gfCNCPoint4[20422] = {X 336.3907, Y 58.0000, Z -6.3333, A 0.000, B 0.000, C 0.000 }
gfCNCPoint4[20423] = {X 336.3907, Y 58.9517, Z -6.3333, A 0.000, B 0.000, C 0.000 }
gfCNCPoint4[20424] = {X 336.3894, Y 59.0936, Z -6.3333, A 0.000, B 0.000, C 0.000 }
gfCNCPoint4[20425] = {X 336.3864, Y 59.2354, Z -6.3333, A 0.000, B 0.000, C 0.000 }
gfCNCPoint4[20426] = {X 336.2429, Y 60.7995, Z -6.3333, A 0.000, B 0.000, C 0.000 }
gfCNCPoint4[20427] = {X 335.8982, Y 62.3319, Z -6.3333, A 0.000, B 0.000, C 0.000 }
gfCNCPoint4[20428] = {X 335.3582, Y 63.8069, Z -6.3333, A 0.000, B 0.000, C 0.000 }
gfCNCPoint4[20429] = {X 334.6320, Y 65.1996, Z -6.3333, A 0.000, B 0.000, C 0.000 }
gfCNCPoint4[20430] = {X 333.7317, Y 66.4867, Z -6.3333, A 0.000, B 0.000, C 0.000 }
gfCNCPoint4[20431] = {X 332.6725, Y 67.6465, Z -6.3333, A 0.000, B 0.000, C 0.000 }
gfCNCPoint4[20432] = {X 332.6738, Y 81.6369, Z -6.3333, A 0.000, B 0.000, C 0.000 }
gfCNCPoint4[20433] = {X 334.6671, Y 81.9567, Z -6.3333, A 0.000, B 0.000, C 0.000 }
gfCNCPoint4[20434] = {X 336.6742, Y 82.1743, Z -6.3333, A 0.000, B 0.000, C 0.000 }
gfCNCPoint4[20435] = {X 340.8156, Y 82.4531, Z -6.3333, A 0.000, B 0.000, C 0.000 }
gfCNCPoint4[20436] = {X 344.9638, Y 82.5981, Z -6.3333, A 0.000, B 0.000, C 0.000 }
gfCNCPoint4[20437] = {X 349.1145, Y 82.6093, Z -6.3333, A 0.000, B 0.000, C 0.000 }
gfCNCPoint4[20438] = {X 353.0020, Y 82.5472, Z -6.3333, A 0.000, B 0.000, C 0.000 }
gfCNCPoint4[20439] = {X 356.8847, Y 82.3434, Z -6.3333, A 0.000, B 0.000, C 0.000 }
gfCNCPoint4[20440] = {X 360.7573, Y 81.9982, Z -6.3333, A 0.000, B 0.000, C 0.000 }
gfCNCPoint4[20441] = {X 361.9619, Y 81.8410, Z -6.3333, A 0.000, B 0.000, C 0.000 }
gfCNCPoint4[20442] = {X 363.1593, Y 81.6353, Z -6.3333, A 0.000, B 0.000, C 0.000 }
gfCNCPoint4[20443] = {X 363.1584, Y 67.6531, Z -6.3333, A 0.000, B 0.000, C 0.000 }
gfCNCPoint4[20444] = {X 362.0724, Y 66.4629, Z -6.3333, A 0.000, B 0.000, C 0.000 }
gfCNCPoint4[20445] = {X 361.1545, Y 65.1387, Z -6.3333, A 0.000, B 0.000, C 0.000 }
gfCNCPoint4[20446] = {X 360.4210, Y 63.7042, Z -6.3333, A 0.000, B 0.000, C 0.000 }
gfCNCPoint4[20447] = {X 359.8849, Y 62.1848, Z -6.3333, A 0.000, B 0.000, C 0.000 }
gfCNCPoint4[20448] = {X 359.5557, Y 60.6075, Z -6.3333, A 0.000, B 0.000, C 0.000 }
gfCNCPoint4[20449] = {X 359.4395, Y 59.0005, Z -6.3333, A 0.000, B 0.000, C 0.000 }
gfCNCPoint4[20450] = {X 359.4393, Y 58.0000, Z -6.3333, A 0.000, B 0.000, C 0.000 }
gfCNCPoint4[20451] = {X 359.5340, Y 56.4902, Z -6.3333, A 0.000, B 0.000, C 0.000 }
gfCNCPoint4[20452] = {X 359.8167, Y 55.0040, Z -6.3333, A 0.000, B 0.000, C 0.000 }
gfCNCPoint4[20453] = {X 359.6068, Y 55.1023, Z -6.3333, A 0.000, B 0.000, C 0.000 }
gfCNCPoint4[20454] = {X 359.3961, Y 55.1989, Z -6.3333, A 0.000, B 0.000, C 0.000 }
gfCNCPoint4[20455] = {X 357.8730, Y 55.8158, Z -6.3333, A 0.000, B 0.000, C 0.000 }
gfCNCPoint4[20456] = {X 356.3192, Y 56.3507, Z -6.3333, A 0.000, B 0.000, C 0.000 }
gfCNCPoint4[20457] = {X 353.9698, Y 56.9888, Z -6.3333, A 0.000, B 0.000, C 0.000 }
gfCNCPoint4[20458] = {X 351.5774, Y 57.4394, Z -6.3333, A 0.000, B 0.000, C 0.000 }
gfCNCPoint4[20459] = {X 349.1568, Y 57.6995, Z -6.3333, A 0.000, B 0.000, C 0.000 }
gfCNCPoint4[20460] = {X 348.9949, Y 55.3050, Z -6.3333, A 0.000, B 0.000, C 0.000 }
gfCNCPoint4[20461] = {X 348.0810, Y 55.3520, Z -6.3333, A 0.000, B 0.000, C 0.000 }
gfCNCPoint4[20462] = {X 347.1660, Y 55.3695, Z -6.3333, A 0.000, B 0.000, C 0.000 }
gfCNCPoint4[20463] = {X 344.5859, Y 55.3176, Z -6.3333, A 0.000, B 0.000, C 0.000 }
gfCNCPoint4[20464] = {X 342.0205, Y 55.0380, Z -6.3333, A 0.000, B 0.000, C 0.000 }
gfCNCPoint4[20465] = {X 339.4899, Y 54.5327, Z -6.3333, A 0.000, B 0.000, C 0.000 }
gfCNCPoint4[20466] = {X 337.0138, Y 53.8057, Z -6.3333, A 0.000, B 0.000, C 0.000 }
gfCNCPoint4[20467] = {X 334.7570, Y 52.9268, Z -6.3333, A 0.000, B 0.000, C 0.000 }
gfCNCPoint4[20468] = {X 332.5808, Y 51.8637, Z -6.3333, A 0.000, B 0.000, C 0.000 }
gfCNCPoint4[20469] = {X 331.5853, Y 51.2779, Z -6.3333, A 0.000, B 0.000, C 0.000 }
gfCNCPoint4[20470] = {X 330.6137, Y 50.6533, Z -6.3333, A 0.000, B 0.000, C 0.000 }
gfCNCPoint4[20471] = {X 331.5795, Y 51.6073, Z -6.3333, A 0.000, B 0.000, C 0.000 }
gfCNCPoint4[20472] = {X 332.4023, Y 52.6870, Z -6.3333, A 0.000, B 0.000, C 0.000 }
gfCNCPoint4[20473] = {X 333.0660, Y 53.8713, Z -6.3333, A 0.000, B 0.000, C 0.000 }
gfCNCPoint4[20474] = {X 333.5575, Y 55.1367, Z -6.3333, A 0.000, B 0.000, C 0.000 }
gfCNCPoint4[20475] = {X 333.8672, Y 56.4585, Z -6.3333, A 0.000, B 0.000, C 0.000 }
gfCNCPoint4[20476] = {X 333.9598, Y 57.2268, Z -6.3333, A 0.000, B 0.000, C 0.000 }
gfCNCPoint4[20477] = {X 333.9907, Y 58.0000, Z -6.3333, A 0.000, B 0.000, C 0.000 }
gfCNCPoint4[20478] = {X 333.9907, Y 58.9439, Z -6.3333, A 0.000, B 0.000, C 0.000 }
gfCNCPoint4[20479] = {X 333.8763, Y 60.3992, Z -6.3333, A 0.000, B 0.000, C 0.000 }
gfCNCPoint4[20480] = {X 333.5452, Y 61.8209, Z -6.3333, A 0.000, B 0.000, C 0.000 }
gfCNCPoint4[20481] = {X 333.0049, Y 63.1770, Z -6.3333, A 0.000, B 0.000, C 0.000 }
gfCNCPoint4[20482] = {X 332.2676, Y 64.4368, Z -6.3333, A 0.000, B 0.000, C 0.000 }
gfCNCPoint4[20483] = {X 331.3498, Y 65.5720, Z -6.3333, A 0.000, B 0.000, C 0.000 }
gfCNCPoint4[20484] = {X 330.2724, Y 66.5569, Z -6.3333, A 0.000, B 0.000, C 0.000 }
gfCNCPoint4[20485] = {X 330.2739, Y 83.2031, Z -6.3333, A 0.000, B 0.000, C 0.000 }
gfCNCPoint4[20486] = {X 330.2776, Y 83.5824, Z -6.3333, A 0.000, B 0.000, C 0.000 }
gfCNCPoint4[20487] = {X 333.3587, Y 84.1905, Z -6.3333, A 0.000, B 0.000, C 0.000 }
gfCNCPoint4[20488] = {X 336.4766, Y 84.5661, Z -6.3333, A 0.000, B 0.000, C 0.000 }
gfCNCPoint4[20489] = {X 340.6882, Y 84.8497, Z -6.3333, A 0.000, B 0.000, C 0.000 }
gfCNCPoint4[20490] = {X 344.9068, Y 84.9975, Z -6.3333, A 0.000, B 0.000, C 0.000 }
gfCNCPoint4[20491] = {X 349.1279, Y 85.0093, Z -6.3333, A 0.000, B 0.000, C 0.000 }
gfCNCPoint4[20492] = {X 353.0977, Y 84.9454, Z -6.3333, A 0.000, B 0.000, C 0.000 }
gfCNCPoint4[20493] = {X 357.0624, Y 84.7369, Z -6.3333, A 0.000, B 0.000, C 0.000 }
gfCNCPoint4[20494] = {X 361.0169, Y 84.3841, Z -6.3333, A 0.000, B 0.000, C 0.000 }
gfCNCPoint4[20495] = {X 363.3029, Y 84.0502, Z -6.3333, A 0.000, B 0.000, C 0.000 }
gfCNCPoint4[20496] = {X 365.5594, Y 83.5549, Z -6.3333, A 0.000, B 0.000, C 0.000 }
gfCNCPoint4[20497] = {X 365.5583, Y 66.5610, Z -6.3333, A 0.000, B 0.000, C 0.000 }
gfCNCPoint4[20498] = {X 364.4841, Y 65.5830, Z -6.3333, A 0.000, B 0.000, C 0.000 }
gfCNCPoint4[20499] = {X 363.5683, Y 64.4553, Z -6.3333, A 0.000, B 0.000, C 0.000 }
gfCNCPoint4[20500] = {X 362.8315, Y 63.2032, Z -6.3333, A 0.000, B 0.000, C 0.000 }
gfCNCPoint4[20501] = {X 362.2905, Y 61.8550, Z -6.3333, A 0.000, B 0.000, C 0.000 }
gfCNCPoint4[20502] = {X 361.9573, Y 60.4410, Z -6.3333, A 0.000, B 0.000, C 0.000 }
gfCNCPoint4[20503] = {X 361.8395, Y 58.9930, Z -6.3333, A 0.000, B 0.000, C 0.000 }
gfCNCPoint4[20504] = {X 361.8393, Y 58.0000, Z -6.3333, A 0.000, B 0.000, C 0.000 }
gfCNCPoint4[20505] = {X 361.9152, Y 56.7901, Z -6.3333, A 0.000, B 0.000, C 0.000 }
gfCNCPoint4[20506] = {X 362.1417, Y 55.5992, Z -6.3333, A 0.000, B 0.000, C 0.000 }
gfCNCPoint4[20507] = {X 362.5727, Y 54.3039, Z -6.3333, A 0.000, B 0.000, C 0.000 }
gfCNCPoint4[20508] = {X 363.1817, Y 53.0820, Z -6.3333, A 0.000, B 0.000, C 0.000 }
gfCNCPoint4[20509] = {X 363.9565, Y 51.9580, Z -6.3333, A 0.000, B 0.000, C 0.000 }
gfCNCPoint4[20510] = {X 364.8817, Y 50.9541, Z -6.3333, A 0.000, B 0.000, C 0.000 }
gfCNCPoint4[20511] = {X 365.9389, Y 50.0904, Z -6.3333, A 0.000, B 0.000, C 0.000 }
gfCNCPoint4[20512] = {X 367.1071, Y 49.3840, Z -6.3333, A 0.000, B 0.000, C 0.000 }
gfCNCPoint4[20513] = {X 368.3631, Y 48.8490, Z -6.3333, A 0.000, B 0.000, C 0.000 }
gfCNCPoint4[20514] = {X 369.6819, Y 48.4960, Z -6.3333, A 0.000, B 0.000, C 0.000 }
gfCNCPoint4[20515] = {X 371.0372, Y 48.3320, Z -6.3333, A 0.000, B 0.000, C 0.000 }
gfCNCPoint4[20516] = {X 371.2782, Y 48.3230, Z -6.3333, A 0.000, B 0.000, C 0.000 }
gfCNCPoint4[20517] = {X 371.5193, Y 48.3200, Z -6.3333, A 0.000, B 0.000, C 0.000 }
gfCNCPoint4[20518] = {X 388.0597, Y 48.3200, Z -6.3333, A 0.000, B 0.000, C 0.000 }
gfCNCPoint4[20519] = {X 389.4419, Y 48.4192, Z -6.3333, A 0.000, B 0.000, C 0.000 }
gfCNCPoint4[20520] = {X 390.7958, Y 48.7147, Z -6.3333, A 0.000, B 0.000, C 0.000 }
gfCNCPoint4[20521] = {X 392.0936, Y 49.2006, Z -6.3333, A 0.000, B 0.000, C 0.000 }
gfCNCPoint4[20522] = {X 393.3087, Y 49.8667, Z -6.3333, A 0.000, B 0.000, C 0.000 }
gfCNCPoint4[20523] = {X 394.5333, Y 49.1962, Z -6.3333, A 0.000, B 0.000, C 0.000 }
gfCNCPoint4[20524] = {X 395.8416, Y 48.7089, Z -6.3333, A 0.000, B 0.000, C 0.000 }
gfCNCPoint4[20525] = {X 397.1858, Y 48.4177, Z -6.3333, A 0.000, B 0.000, C 0.000 }
gfCNCPoint4[20526] = {X 398.5577, Y 48.3200, Z -6.3333, A 0.000, B 0.000, C 0.000 }
gfCNCPoint4[20527] = {X 398.7346, Y 48.3200, Z -6.3333, A 0.000, B 0.000, C 0.000 }
gfCNCPoint4[20528] = {X 398.1859, Y 47.6069, Z -6.3333, A 0.000, B 0.000, C 0.000 }
gfCNCPoint4[20529] = {X 397.7774, Y 46.8051, Z -6.3333, A 0.000, B 0.000, C 0.000 }
gfCNCPoint4[20530] = {X 397.5230, Y 45.9420, Z -6.3333, A 0.000, B 0.000, C 0.000 }
gfCNCPoint4[20531] = {X 397.4561, Y 45.4921, Z -6.3333, A 0.000, B 0.000, C 0.000 }
gfCNCPoint4[20532] = {X 397.4314, Y 45.0378, Z -6.3333, A 0.000, B 0.000, C 0.000 }
gfCNCPoint4[20533] = {X 397.4316, Y 44.1456, Z -6.3333, A 0.000, B 0.000, C 0.000 }
gfCNCPoint4[20534] = {X 397.5413, Y 43.1780, Z -6.3333, A 0.000, B 0.000, C 0.000 }
gfCNCPoint4[20535] = {X 397.8410, Y 42.2514, Z -6.3333, A 0.000, B 0.000, C 0.000 }
gfCNCPoint4[20536] = {X 398.3186, Y 41.4029, Z -6.3333, A 0.000, B 0.000, C 0.000 }
gfCNCPoint4[20537] = {X 398.9552, Y 40.6660, Z -6.3333, A 0.000, B 0.000, C 0.000 }
gfCNCPoint4[20538] = {X 398.9552, Y 31.8248, Z -6.3333, A 0.000, B 0.000, C 0.000 }
gfCNCPoint4[20539] = {X 396.7504, Y 27.9907, Z -6.3333, A 0.000, B 0.000, C 0.000 }
gfCNCPoint4[20540] = {X 386.3478, Y 33.9728, Z -6.3333, A 0.000, B 0.000, C 0.000 }
gfCNCPoint4[20541] = {X 386.2674, Y 34.3975, Z -6.3333, A 0.000, B 0.000, C 0.000 }
gfCNCPoint4[20542] = {X 386.1833, Y 34.8215, Z -6.3333, A 0.000, B 0.000, C 0.000 }
gfCNCPoint4[20543] = {X 386.0240, Y 35.5723, Z -6.3333, A 0.000, B 0.000, C 0.000 }
gfCNCPoint4[20544] = {X 385.8510, Y 36.3200, Z -6.3333, A 0.000, B 0.000, C 0.000 }
gfCNCPoint4[20545] = {X 386.9552, Y 36.3200, Z -6.3333, A 0.000, B 0.000, C 0.000 }
gfCNCPoint4[20546] = {X 386.9552, Y 35.0290, Z -6.3333, A 0.000, B 0.000, C 0.000 }
gfCNCPoint4[20547] = {X 386.3478, Y 33.9728, Z -6.3333, A 0.000, B 0.000, C 0.000 }
gfCNCPoint4[20548] = {X 388.4283, Y 32.7764, Z -6.3333, A 0.000, B 0.000, C 0.000 }
gfCNCPoint4[20549] = {X 384.7454, Y 26.3718, Z -6.3333, A 0.000, B 0.000, C 0.000 }
gfCNCPoint4[20550] = {X 384.6159, Y 28.7722, Z -6.3333, A 0.000, B 0.000, C 0.000 }
gfCNCPoint4[20551] = {X 384.3631, Y 31.1627, Z -6.3333, A 0.000, B 0.000, C 0.000 }
gfCNCPoint4[20552] = {X 383.9877, Y 33.5370, Z -6.3333, A 0.000, B 0.000, C 0.000 }
gfCNCPoint4[20553] = {X 383.9112, Y 33.9411, Z -6.3333, A 0.000, B 0.000, C 0.000 }
gfCNCPoint4[20554] = {X 383.8312, Y 34.3445, Z -6.3333, A 0.000, B 0.000, C 0.000 }
gfCNCPoint4[20555] = {X 383.6810, Y 35.0524, Z -6.3333, A 0.000, B 0.000, C 0.000 }
gfCNCPoint4[20556] = {X 383.5178, Y 35.7575, Z -6.3333, A 0.000, B 0.000, C 0.000 }
gfCNCPoint4[20557] = {X 383.1278, Y 37.2469, Z -6.3333, A 0.000, B 0.000, C 0.000 }
gfCNCPoint4[20558] = {X 382.6801, Y 38.7200, Z -6.3333, A 0.000, B 0.000, C 0.000 }
gfCNCPoint4[20559] = {X 388.0597, Y 38.7200, Z -6.3333, A 0.000, B 0.000, C 0.000 }
gfCNCPoint4[20560] = {X 388.4821, Y 38.7246, Z -6.3333, A 0.000, B 0.000, C 0.000 }
gfCNCPoint4[20561] = {X 388.9042, Y 38.7385, Z -6.3333, A 0.000, B 0.000, C 0.000 }
gfCNCPoint4[20562] = {X 389.1203, Y 38.2363, Z -6.3333, A 0.000, B 0.000, C 0.000 }
gfCNCPoint4[20563] = {X 389.3552, Y 37.7426, Z -6.3333, A 0.000, B 0.000, C 0.000 }
gfCNCPoint4[20564] = {X 389.3552, Y 34.3882, Z -6.3333, A 0.000, B 0.000, C 0.000 }
gfCNCPoint4[20565] = {X 388.4283, Y 32.7764, Z -6.3333, A 0.000, B 0.000, C 0.000 }
gfCNCPoint4[20566] = {X 390.5088, Y 31.5799, Z -6.3333, A 0.000, B 0.000, C 0.000 }
gfCNCPoint4[20567] = {X 386.7932, Y 25.1185, Z -6.3333, A 0.000, B 0.000, C 0.000 }
gfCNCPoint4[20568] = {X 386.1529, Y 24.0242, Z -6.3333, A 0.000, B 0.000, C 0.000 }
gfCNCPoint4[20569] = {X 385.4963, Y 22.9396, Z -6.3333, A 0.000, B 0.000, C 0.000 }
gfCNCPoint4[20570] = {X 384.4704, Y 22.1518, Z -6.3333, A 0.000, B 0.000, C 0.000 }
gfCNCPoint4[20571] = {X 383.5345, Y 21.2589, Z -6.3333, A 0.000, B 0.000, C 0.000 }
gfCNCPoint4[20572] = {X 382.6995, Y 20.2710, Z -6.3333, A 0.000, B 0.000, C 0.000 }
gfCNCPoint4[20573] = {X 381.9749, Y 19.1995, Z -6.3333, A 0.000, B 0.000, C 0.000 }
gfCNCPoint4[20574] = {X 382.2256, Y 21.5600, Z -6.3333, A 0.000, B 0.000, C 0.000 }
gfCNCPoint4[20575] = {X 382.3495, Y 23.9305, Z -6.3333, A 0.000, B 0.000, C 0.000 }
gfCNCPoint4[20576] = {X 382.3463, Y 26.3043, Z -6.3333, A 0.000, B 0.000, C 0.000 }
gfCNCPoint4[20577] = {X 382.2021, Y 28.8406, Z -6.3333, A 0.000, B 0.000, C 0.000 }
gfCNCPoint4[20578] = {X 381.9127, Y 31.3644, Z -6.3333, A 0.000, B 0.000, C 0.000 }
gfCNCPoint4[20579] = {X 381.4791, Y 33.8675, Z -6.3333, A 0.000, B 0.000, C 0.000 }
gfCNCPoint4[20580] = {X 380.9974, Y 35.9380, Z -6.3333, A 0.000, B 0.000, C 0.000 }
gfCNCPoint4[20581] = {X 380.3978, Y 37.9774, Z -6.3333, A 0.000, B 0.000, C 0.000 }
gfCNCPoint4[20582] = {X 379.8422, Y 39.5621, Z -6.3333, A 0.000, B 0.000, C 0.000 }
gfCNCPoint4[20583] = {X 379.2155, Y 41.1200, Z -6.3333, A 0.000, B 0.000, C 0.000 }
gfCNCPoint4[20584] = {X 388.0597, Y 41.1200, Z -6.3333, A 0.000, B 0.000, C 0.000 }
gfCNCPoint4[20585] = {X 389.3255, Y 41.1675, Z -6.3333, A 0.000, B 0.000, C 0.000 }
gfCNCPoint4[20586] = {X 390.5842, Y 41.3098, Z -6.3333, A 0.000, B 0.000, C 0.000 }
gfCNCPoint4[20587] = {X 391.0709, Y 39.7837, Z -6.3333, A 0.000, B 0.000, C 0.000 }
gfCNCPoint4[20588] = {X 391.7552, Y 38.3354, Z -6.3333, A 0.000, B 0.000, C 0.000 }
gfCNCPoint4[20589] = {X 391.7552, Y 33.7473, Z -6.3333, A 0.000, B 0.000, C 0.000 }
gfCNCPoint4[20590] = {X 390.5088, Y 31.5799, Z -6.3333, A 0.000, B 0.000, C 0.000 }
gfCNCPoint4[20591] = {X 392.5894, Y 30.3835, Z -6.3333, A 0.000, B 0.000, C 0.000 }
gfCNCPoint4[20592] = {X 388.8737, Y 23.9221, Z -6.3333, A 0.000, B 0.000, C 0.000 }
gfCNCPoint4[20593] = {X 388.0764, Y 22.5642, Z -6.3333, A 0.000, B 0.000, C 0.000 }
gfCNCPoint4[20594] = {X 387.2547, Y 21.2210, Z -6.3333, A 0.000, B 0.000, C 0.000 }
gfCNCPoint4[20595] = {X 386.3084, Y 20.5574, Z -6.3333, A 0.000, B 0.000, C 0.000 }
gfCNCPoint4[20596] = {X 385.4479, Y 19.7857, Z -6.3333, A 0.000, B 0.000, C 0.000 }
gfCNCPoint4[20597] = {X 384.6855, Y 18.9169, Z -6.3333, A 0.000, B 0.000, C 0.000 }
gfCNCPoint4[20598] = {X 384.0321, Y 17.9634, Z -6.3333, A 0.000, B 0.000, C 0.000 }
gfCNCPoint4[20599] = {X 383.4422, Y 16.8142, Z -6.3333, A 0.000, B 0.000, C 0.000 }
gfCNCPoint4[20600] = {X 383.0106, Y 15.5967, Z -6.3333, A 0.000, B 0.000, C 0.000 }
gfCNCPoint4[20601] = {X 382.7449, Y 14.3326, Z -6.3333, A 0.000, B 0.000, C 0.000 }
gfCNCPoint4[20602] = {X 382.6498, Y 13.0443, Z -6.3333, A 0.000, B 0.000, C 0.000 }
gfCNCPoint4[20603] = {X 382.6496, Y 12.1868, Z -6.3333, A 0.000, B 0.000, C 0.000 }
gfCNCPoint4[20604] = {X 382.6507, Y 12.0458, Z -6.3333, A 0.000, B 0.000, C 0.000 }
gfCNCPoint4[20605] = {X 382.6537, Y 11.9049, Z -6.3333, A 0.000, B 0.000, C 0.000 }
gfCNCPoint4[20606] = {X 377.7904, Y 11.9049, Z -6.3333, A 0.000, B 0.000, C 0.000 }
gfCNCPoint4[20607] = {X 378.4102, Y 13.8166, Z -6.3333, A 0.000, B 0.000, C 0.000 }
gfCNCPoint4[20608] = {X 378.9201, Y 15.7606, Z -6.3333, A 0.000, B 0.000, C 0.000 }
gfCNCPoint4[20609] = {X 379.3184, Y 17.7304, Z -6.3333, A 0.000, B 0.000, C 0.000 }
gfCNCPoint4[20610] = {X 379.4668, Y 18.6221, Z -6.3333, A 0.000, B 0.000, C 0.000 }
gfCNCPoint4[20611] = {X 379.5960, Y 19.5168, Z -6.3333, A 0.000, B 0.000, C 0.000 }
gfCNCPoint4[20612] = {X 379.8725, Y 22.2917, Z -6.3333, A 0.000, B 0.000, C 0.000 }
gfCNCPoint4[20613] = {X 379.9639, Y 25.0789, Z -6.3333, A 0.000, B 0.000, C 0.000 }
gfCNCPoint4[20614] = {X 379.8697, Y 27.8660, Z -6.3333, A 0.000, B 0.000, C 0.000 }
gfCNCPoint4[20615] = {X 379.5903, Y 30.6407, Z -6.3333, A 0.000, B 0.000, C 0.000 }
gfCNCPoint4[20616] = {X 379.1270, Y 33.3906, Z -6.3333, A 0.000, B 0.000, C 0.000 }
gfCNCPoint4[20617] = {X 378.5766, Y 35.6983, Z -6.3333, A 0.000, B 0.000, C 0.000 }
gfCNCPoint4[20618] = {X 377.8697, Y 37.9630, Z -6.3333, A 0.000, B 0.000, C 0.000 }
gfCNCPoint4[20619] = {X 377.0098, Y 40.1741, Z -6.3333, A 0.000, B 0.000, C 0.000 }
gfCNCPoint4[20620] = {X 376.2281, Y 41.8693, Z -6.3333, A 0.000, B 0.000, C 0.000 }
gfCNCPoint4[20621] = {X 375.3564, Y 43.5200, Z -6.3333, A 0.000, B 0.000, C 0.000 }
gfCNCPoint4[20622] = {X 388.0597, Y 43.5200, Z -6.3333, A 0.000, B 0.000, C 0.000 }
gfCNCPoint4[20623] = {X 389.6072, Y 43.6029, Z -6.3333, A 0.000, B 0.000, C 0.000 }
gfCNCPoint4[20624] = {X 391.1370, Y 43.8508, Z -6.3333, A 0.000, B 0.000, C 0.000 }
gfCNCPoint4[20625] = {X 392.6316, Y 44.2607, Z -6.3333, A 0.000, B 0.000, C 0.000 }
gfCNCPoint4[20626] = {X 392.6316, Y 44.1162, Z -6.3333, A 0.000, B 0.000, C 0.000 }
gfCNCPoint4[20627] = {X 392.7390, Y 42.7683, Z -6.3333, A 0.000, B 0.000, C 0.000 }
gfCNCPoint4[20628] = {X 393.0331, Y 41.4485, Z -6.3333, A 0.000, B 0.000, C 0.000 }
gfCNCPoint4[20629] = {X 393.5083, Y 40.1826, Z -6.3333, A 0.000, B 0.000, C 0.000 }
gfCNCPoint4[20630] = {X 394.1552, Y 38.9952, Z -6.3333, A 0.000, B 0.000, C 0.000 }
gfCNCPoint4[20631] = {X 394.1552, Y 33.1065, Z -6.3333, A 0.000, B 0.000, C 0.000 }
gfCNCPoint4[20632] = {X 392.5894, Y 30.3835, Z -6.3333, A 0.000, B 0.000, C 0.000 }
gfCNCPoint4[20633] = {X 394.6699, Y 29.1871, Z -6.3333, A 0.000, B 0.000, C 0.000 }
gfCNCPoint4[20634] = {X 390.9542, Y 22.7257, Z -6.3333, A 0.000, B 0.000, C 0.000 }
gfCNCPoint4[20635] = {X 390.0941, Y 21.2622, Z -6.3333, A 0.000, B 0.000, C 0.000 }
gfCNCPoint4[20636] = {X 389.2063, Y 19.8154, Z -6.3333, A 0.000, B 0.000, C 0.000 }
gfCNCPoint4[20637] = {X 389.0623, Y 19.6029, Z -6.3333, A 0.000, B 0.000, C 0.000 }
gfCNCPoint4[20638] = {X 388.9034, Y 19.4014, Z -6.3333, A 0.000, B 0.000, C 0.000 }
gfCNCPoint4[20639] = {X 387.8155, Y 18.6895, Z -6.3333, A 0.000, B 0.000, C 0.000 }
gfCNCPoint4[20640] = {X 386.8715, Y 17.7954, Z -6.3333, A 0.000, B 0.000, C 0.000 }
gfCNCPoint4[20641] = {X 386.1016, Y 16.7477, Z -6.3333, A 0.000, B 0.000, C 0.000 }
gfCNCPoint4[20642] = {X 385.5304, Y 15.5797, Z -6.3333, A 0.000, B 0.000, C 0.000 }
gfCNCPoint4[20643] = {X 385.1760, Y 14.3287, Z -6.3333, A 0.000, B 0.000, C 0.000 }
gfCNCPoint4[20644] = {X 385.0498, Y 13.0347, Z -6.3333, A 0.000, B 0.000, C 0.000 }
gfCNCPoint4[20645] = {X 385.0496, Y 12.1868, Z -6.3333, A 0.000, B 0.000, C 0.000 }
gfCNCPoint4[20646] = {X 385.0504, Y 12.0808, Z -6.3333, A 0.000, B 0.000, C 0.000 }
gfCNCPoint4[20647] = {X 385.0527, Y 11.9748, Z -6.3333, A 0.000, B 0.000, C 0.000 }
gfCNCPoint4[20648] = {X 385.1994, Y 10.7176, Z -6.3333, A 0.000, B 0.000, C 0.000 }
gfCNCPoint4[20649] = {X 385.5616, Y 9.5049, Z -6.3333, A 0.000, B 0.000, C 0.000 }
gfCNCPoint4[20650] = {X 374.1938, Y 9.5049, Z -6.3333, A 0.000, B 0.000, C 0.000 }
gfCNCPoint4[20651] = {X 374.9040, Y 11.0897, Z -6.3333, A 0.000, B 0.000, C 0.000 }
gfCNCPoint4[20652] = {X 375.5294, Y 12.7098, Z -6.3333, A 0.000, B 0.000, C 0.000 }
gfCNCPoint4[20653] = {X 376.1076, Y 14.4932, Z -6.3333, A 0.000, B 0.000, C 0.000 }
gfCNCPoint4[20654] = {X 376.5831, Y 16.3068, Z -6.3333, A 0.000, B 0.000, C 0.000 }
gfCNCPoint4[20655] = {X 376.9543, Y 18.1444, Z -6.3333, A 0.000, B 0.000, C 0.000 }
gfCNCPoint4[20656] = {X 377.3638, Y 21.0869, Z -6.3333, A 0.000, B 0.000, C 0.000 }
gfCNCPoint4[20657] = {X 377.5511, Y 24.0518, Z -6.3333, A 0.000, B 0.000, C 0.000 }
gfCNCPoint4[20658] = {X 377.5150, Y 27.0224, Z -6.3333, A 0.000, B 0.000, C 0.000 }
gfCNCPoint4[20659] = {X 377.2557, Y 29.9819, Z -6.3333, A 0.000, B 0.000, C 0.000 }
gfCNCPoint4[20660] = {X 376.7748, Y 32.9136, Z -6.3333, A 0.000, B 0.000, C 0.000 }
gfCNCPoint4[20661] = {X 376.1771, Y 35.3667, Z -6.3333, A 0.000, B 0.000, C 0.000 }
gfCNCPoint4[20662] = {X 375.3894, Y 37.7656, Z -6.3333, A 0.000, B 0.000, C 0.000 }
gfCNCPoint4[20663] = {X 374.4168, Y 40.0957, Z -6.3333, A 0.000, B 0.000, C 0.000 }
gfCNCPoint4[20664] = {X 373.2651, Y 42.3426, Z -6.3333, A 0.000, B 0.000, C 0.000 }
gfCNCPoint4[20665] = {X 372.1957, Y 44.1076, Z -6.3333, A 0.000, B 0.000, C 0.000 }
gfCNCPoint4[20666] = {X 371.0159, Y 45.8006, Z -6.3333, A 0.000, B 0.000, C 0.000 }
gfCNCPoint4[20667] = {X 370.9177, Y 45.9350, Z -6.3333, A 0.000, B 0.000, C 0.000 }
gfCNCPoint4[20668] = {X 371.2184, Y 45.9237, Z -6.3333, A 0.000, B 0.000, C 0.000 }
gfCNCPoint4[20669] = {X 371.5193, Y 45.9200, Z -6.3333, A 0.000, B 0.000, C 0.000 }
gfCNCPoint4[20670] = {X 388.0597, Y 45.9200, Z -6.3333, A 0.000, B 0.000, C 0.000 }
gfCNCPoint4[20671] = {X 389.4143, Y 45.9962, Z -6.3333, A 0.000, B 0.000, C 0.000 }
gfCNCPoint4[20672] = {X 390.7519, Y 46.2238, Z -6.3333, A 0.000, B 0.000, C 0.000 }
gfCNCPoint4[20673] = {X 392.0555, Y 46.6000, Z -6.3333, A 0.000, B 0.000, C 0.000 }
gfCNCPoint4[20674] = {X 393.3087, Y 47.1200, Z -6.3333, A 0.000, B 0.000, C 0.000 }
gfCNCPoint4[20675] = {X 394.2237, Y 46.7243, Z -6.3333, A 0.000, B 0.000, C 0.000 }
gfCNCPoint4[20676] = {X 395.1681, Y 46.4053, Z -6.3333, A 0.000, B 0.000, C 0.000 }
gfCNCPoint4[20677] = {X 395.0678, Y 45.7292, Z -6.3333, A 0.000, B 0.000, C 0.000 }
gfCNCPoint4[20678] = {X 395.0314, Y 45.0468, Z -6.3333, A 0.000, B 0.000, C 0.000 }
gfCNCPoint4[20679] = {X 395.0316, Y 44.1297, Z -6.3333, A 0.000, B 0.000, C 0.000 }
gfCNCPoint4[20680] = {X 395.1397, Y 42.9565, Z -6.3333, A 0.000, B 0.000, C 0.000 }
gfCNCPoint4[20681] = {X 395.4356, Y 41.8161, Z -6.3333, A 0.000, B 0.000, C 0.000 }
gfCNCPoint4[20682] = {X 395.9116, Y 40.7384, Z -6.3333, A 0.000, B 0.000, C 0.000 }
gfCNCPoint4[20683] = {X 396.5552, Y 39.7516, Z -6.3333, A 0.000, B 0.000, C 0.000 }
gfCNCPoint4[20684] = {X 396.5552, Y 32.4656, Z -6.3333, A 0.000, B 0.000, C 0.000 }
gfCNCPoint4[20685] = {X 394.6699, Y 29.1871, Z -6.3333, A 0.000, B 0.000, C 0.000 }
gfCNCPoint4[20686] = {X 396.7504, Y 27.9907, Z -6.3333, A 0.000, B 0.000, C 0.000 }
gfCNCPoint4[20687] = {X 393.0348, Y 21.5292, Z -6.3333, A 0.000, B 0.000, C 0.000 }
gfCNCPoint4[20688] = {X 392.1515, Y 20.0265, Z -6.3333, A 0.000, B 0.000, C 0.000 }
gfCNCPoint4[20689] = {X 391.2398, Y 18.5408, Z -6.3333, A 0.000, B 0.000, C 0.000 }
gfCNCPoint4[20690] = {X 390.8286, Y 17.9637, Z -6.3333, A 0.000, B 0.000, C 0.000 }
gfCNCPoint4[20691] = {X 390.3520, Y 17.4394, Z -6.3333, A 0.000, B 0.000, C 0.000 }
gfCNCPoint4[20692] = {X 389.5422, Y 16.9836, Z -6.3333, A 0.000, B 0.000, C 0.000 }
gfCNCPoint4[20693] = {X 388.8334, Y 16.3826, Z -6.3333, A 0.000, B 0.000, C 0.000 }
gfCNCPoint4[20694] = {X 388.2515, Y 15.6581, Z -6.3333, A 0.000, B 0.000, C 0.000 }
gfCNCPoint4[20695] = {X 387.8174, Y 14.8365, Z -6.3333, A 0.000, B 0.000, C 0.000 }
gfCNCPoint4[20696] = {X 387.5469, Y 13.9474, Z -6.3333, A 0.000, B 0.000, C 0.000 }
gfCNCPoint4[20697] = {X 387.4498, Y 13.0232, Z -6.3333, A 0.000, B 0.000, C 0.000 }
gfCNCPoint4[20698] = {X 387.4496, Y 12.1868, Z -6.3333, A 0.000, B 0.000, C 0.000 }
gfCNCPoint4[20699] = {X 387.5362, Y 11.2717, Z -6.3333, A 0.000, B 0.000, C 0.000 }
gfCNCPoint4[20700] = {X 387.7928, Y 10.3890, Z -6.3333, A 0.000, B 0.000, C 0.000 }
gfCNCPoint4[20701] = {X 388.2376, Y 9.5280, Z -6.3333, A 0.000, B 0.000, C 0.000 }
gfCNCPoint4[20702] = {X 388.8437, Y 8.7718, Z -6.3333, A 0.000, B 0.000, C 0.000 }
gfCNCPoint4[20703] = {X 389.5873, Y 8.1503, Z -6.3333, A 0.000, B 0.000, C 0.000 }
gfCNCPoint4[20704] = {X 390.4390, Y 7.6879, Z -6.3333, A 0.000, B 0.000, C 0.000 }
gfCNCPoint4[20705] = {X 391.3653, Y 7.4030, Z -6.3333, A 0.000, B 0.000, C 0.000 }
gfCNCPoint4[20706] = {X 392.3296, Y 7.3068, Z -6.3333, A 0.000, B 0.000, C 0.000 }
gfCNCPoint4[20707] = {X 399.1118, Y 7.3068, Z -6.3333, A 0.000, B 0.000, C 0.000 }
gfCNCPoint4[20708] = {X 400.0638, Y 7.4006, Z -6.3333, A 0.000, B 0.000, C 0.000 }
gfCNCPoint4[20709] = {X 400.9793, Y 7.6783, Z -6.3333, A 0.000, B 0.000, C 0.000 }
gfCNCPoint4[20710] = {X 401.8229, Y 8.1292, Z -6.3333, A 0.000, B 0.000, C 0.000 }
gfCNCPoint4[20711] = {X 402.5624, Y 8.7361, Z -6.3333, A 0.000, B 0.000, C 0.000 }
gfCNCPoint4[20712] = {X 403.1693, Y 9.4756, Z -6.3333, A 0.000, B 0.000, C 0.000 }
gfCNCPoint4[20713] = {X 403.6203, Y 10.3193, Z -6.3333, A 0.000, B 0.000, C 0.000 }
gfCNCPoint4[20714] = {X 403.8980, Y 11.2348, Z -6.3333, A 0.000, B 0.000, C 0.000 }
gfCNCPoint4[20715] = {X 403.9918, Y 12.1868, Z -6.3333, A 0.000, B 0.000, C 0.000 }
gfCNCPoint4[20716] = {X 403.9915, Y 13.0237, Z -6.3333, A 0.000, B 0.000, C 0.000 }
gfCNCPoint4[20717] = {X 403.9016, Y 13.9115, Z -6.3333, A 0.000, B 0.000, C 0.000 }
gfCNCPoint4[20718] = {X 403.6516, Y 14.7680, Z -6.3333, A 0.000, B 0.000, C 0.000 }
gfCNCPoint4[20719] = {X 405.3644, Y 17.7421, Z -6.3333, A 0.000, B 0.000, C 0.000 }
gfCNCPoint4[20720] = {X 407.2444, Y 14.6971, Z -6.3333, A 0.000, B 0.000, C 0.000 }
gfCNCPoint4[20721] = {X 407.0142, Y 13.8723, Z -6.3333, A 0.000, B 0.000, C 0.000 }
gfCNCPoint4[20722] = {X 406.9317, Y 13.0199, Z -6.3333, A 0.000, B 0.000, C 0.000 }
gfCNCPoint4[20723] = {X 406.9315, Y 12.1868, Z -6.3333, A 0.000, B 0.000, C 0.000 }
gfCNCPoint4[20724] = {X 407.0253, Y 11.2348, Z -6.3333, A 0.000, B 0.000, C 0.000 }
gfCNCPoint4[20725] = {X 407.3030, Y 10.3193, Z -6.3333, A 0.000, B 0.000, C 0.000 }
gfCNCPoint4[20726] = {X 407.7540, Y 9.4756, Z -6.3333, A 0.000, B 0.000, C 0.000 }
gfCNCPoint4[20727] = {X 408.3609, Y 8.7361, Z -6.3333, A 0.000, B 0.000, C 0.000 }
gfCNCPoint4[20728] = {X 409.1004, Y 8.1292, Z -6.3333, A 0.000, B 0.000, C 0.000 }
gfCNCPoint4[20729] = {X 409.9440, Y 7.6783, Z -6.3333, A 0.000, B 0.000, C 0.000 }
gfCNCPoint4[20730] = {X 410.8595, Y 7.4006, Z -6.3333, A 0.000, B 0.000, C 0.000 }
gfCNCPoint4[20731] = {X 411.8115, Y 7.3068, Z -6.3333, A 0.000, B 0.000, C 0.000 }
gfCNCPoint4[20732] = {X 419.3245, Y 7.3068, Z -6.3333, A 0.000, B 0.000, C 0.000 }
gfCNCPoint4[20733] = {X 420.2888, Y 7.4030, Z -6.3333, A 0.000, B 0.000, C 0.000 }
gfCNCPoint4[20734] = {X 421.2151, Y 7.6879, Z -6.3333, A 0.000, B 0.000, C 0.000 }
gfCNCPoint4[20735] = {X 422.0668, Y 8.1503, Z -6.3333, A 0.000, B 0.000, C 0.000 }
gfCNCPoint4[20736] = {X 422.8104, Y 8.7718, Z -6.3333, A 0.000, B 0.000, C 0.000 }
gfCNCPoint4[20737] = {X 423.4165, Y 9.5280, Z -6.3333, A 0.000, B 0.000, C 0.000 }
gfCNCPoint4[20738] = {X 423.8612, Y 10.3890, Z -6.3333, A 0.000, B 0.000, C 0.000 }
gfCNCPoint4[20739] = {X 424.1179, Y 11.2717, Z -6.3333, A 0.000, B 0.000, C 0.000 }
gfCNCPoint4[20740] = {X 424.2045, Y 12.1868, Z -6.3333, A 0.000, B 0.000, C 0.000 }
gfCNCPoint4[20741] = {X 424.2045, Y 12.9780, Z -6.3333, A 0.000, B 0.000, C 0.000 }
gfCNCPoint4[20742] = {X 424.1063, Y 13.9308, Z -6.3333, A 0.000, B 0.000, C 0.000 }
gfCNCPoint4[20743] = {X 423.8261, Y 14.8468, Z -6.3333, A 0.000, B 0.000, C 0.000 }
gfCNCPoint4[20744] = {X 423.3745, Y 15.6915, Z -6.3333, A 0.000, B 0.000, C 0.000 }
gfCNCPoint4[20745] = {X 422.7684, Y 16.4332, Z -6.3333, A 0.000, B 0.000, C 0.000 }
gfCNCPoint4[20746] = {X 422.0306, Y 17.0441, Z -6.3333, A 0.000, B 0.000, C 0.000 }
gfCNCPoint4[20747] = {X 421.1888, Y 17.5011, Z -6.3333, A 0.000, B 0.000, C 0.000 }
gfCNCPoint4[20748] = {X 420.5409, Y 18.3845, Z -6.3333, A 0.000, B 0.000, C 0.000 }
gfCNCPoint4[20749] = {X 419.9519, Y 19.3082, Z -6.3333, A 0.000, B 0.000, C 0.000 }
gfCNCPoint4[20750] = {X 414.1625, Y 28.6201, Z -6.3333, A 0.000, B 0.000, C 0.000 }
gfCNCPoint4[20751] = {X 422.3153, Y 33.6888, Z -6.3333, A 0.000, B 0.000, C 0.000 }
gfCNCPoint4[20752] = {X 421.8946, Y 34.3655, Z -6.3333, A 0.000, B 0.000, C 0.000 }
gfCNCPoint4[20753] = {X 422.1476, Y 34.0994, Z -6.3333, A 0.000, B 0.000, C 0.000 }
gfCNCPoint4[20754] = {X 422.4073, Y 33.8398, Z -6.3333, A 0.000, B 0.000, C 0.000 }
gfCNCPoint4[20755] = {X 422.3611, Y 33.7644, Z -6.3333, A 0.000, B 0.000, C 0.000 }
gfCNCPoint4[20756] = {X 422.3153, Y 33.6888, Z -6.3333, A 0.000, B 0.000, C 0.000 }
gfCNCPoint4[20757] = {X 420.2771, Y 32.4217, Z -6.3333, A 0.000, B 0.000, C 0.000 }
gfCNCPoint4[20758] = {X 419.3077, Y 33.9809, Z -6.3333, A 0.000, B 0.000, C 0.000 }
gfCNCPoint4[20759] = {X 419.3080, Y 38.3386, Z -6.3333, A 0.000, B 0.000, C 0.000 }
gfCNCPoint4[20760] = {X 419.9584, Y 39.7075, Z -6.3333, A 0.000, B 0.000, C 0.000 }
gfCNCPoint4[20761] = {X 420.4340, Y 41.1465, Z -6.3333, A 0.000, B 0.000, C 0.000 }
gfCNCPoint4[20762] = {X 420.6282, Y 41.1585, Z -6.3333, A 0.000, B 0.000, C 0.000 }
gfCNCPoint4[20763] = {X 420.8222, Y 41.1728, Z -6.3333, A 0.000, B 0.000, C 0.000 }
gfCNCPoint4[20764] = {X 421.2846, Y 39.7572, Z -6.3333, A 0.000, B 0.000, C 0.000 }
gfCNCPoint4[20765] = {X 421.9176, Y 38.4093, Z -6.3333, A 0.000, B 0.000, C 0.000 }
gfCNCPoint4[20766] = {X 422.7117, Y 37.1495, Z -6.3333, A 0.000, B 0.000, C 0.000 }
gfCNCPoint4[20767] = {X 423.6548, Y 35.9970, Z -6.3333, A 0.000, B 0.000, C 0.000 }
gfCNCPoint4[20768] = {X 424.3425, Y 35.3124, Z -6.3333, A 0.000, B 0.000, C 0.000 }
gfCNCPoint4[20769] = {X 425.0829, Y 34.6852, Z -6.3333, A 0.000, B 0.000, C 0.000 }
gfCNCPoint4[20770] = {X 425.4252, Y 34.0151, Z -6.3333, A 0.000, B 0.000, C 0.000 }
gfCNCPoint4[20771] = {X 424.8781, Y 33.2447, Z -6.3333, A 0.000, B 0.000, C 0.000 }
gfCNCPoint4[20772] = {X 424.3698, Y 32.4482, Z -6.3333, A 0.000, B 0.000, C 0.000 }
gfCNCPoint4[20773] = {X 423.3888, Y 30.6023, Z -6.3333, A 0.000, B 0.000, C 0.000 }
gfCNCPoint4[20774] = {X 422.6157, Y 28.6601, Z -6.3333, A 0.000, B 0.000, C 0.000 }
gfCNCPoint4[20775] = {X 420.2771, Y 32.4217, Z -6.3333, A 0.000, B 0.000, C 0.000 }
gfCNCPoint4[20776] = {X 418.2389, Y 31.1545, Z -6.3333, A 0.000, B 0.000, C 0.000 }
gfCNCPoint4[20777] = {X 416.9077, Y 33.2957, Z -6.3333, A 0.000, B 0.000, C 0.000 }
gfCNCPoint4[20778] = {X 416.9081, Y 38.9952, Z -6.3333, A 0.000, B 0.000, C 0.000 }
gfCNCPoint4[20779] = {X 417.4894, Y 40.0484, Z -6.3333, A 0.000, B 0.000, C 0.000 }
gfCNCPoint4[20780] = {X 417.9372, Y 41.1650, Z -6.3333, A 0.000, B 0.000, C 0.000 }
gfCNCPoint4[20781] = {X 418.2449, Y 42.3280, Z -6.3333, A 0.000, B 0.000, C 0.000 }
gfCNCPoint4[20782] = {X 418.4078, Y 43.5200, Z -6.3333, A 0.000, B 0.000, C 0.000 }
gfCNCPoint4[20783] = {X 419.4886, Y 43.5200, Z -6.3333, A 0.000, B 0.000, C 0.000 }
gfCNCPoint4[20784] = {X 421.1752, Y 43.6186, Z -6.3333, A 0.000, B 0.000, C 0.000 }
gfCNCPoint4[20785] = {X 422.8389, Y 43.9129, Z -6.3333, A 0.000, B 0.000, C 0.000 }
gfCNCPoint4[20786] = {X 423.0005, Y 42.4234, Z -6.3333, A 0.000, B 0.000, C 0.000 }
gfCNCPoint4[20787] = {X 423.3900, Y 40.9766, Z -6.3333, A 0.000, B 0.000, C 0.000 }
gfCNCPoint4[20788] = {X 423.9980, Y 39.6073, Z -6.3333, A 0.000, B 0.000, C 0.000 }
gfCNCPoint4[20789] = {X 424.8102, Y 38.3482, Z -6.3333, A 0.000, B 0.000, C 0.000 }
gfCNCPoint4[20790] = {X 425.8068, Y 37.2295, Z -6.3333, A 0.000, B 0.000, C 0.000 }
gfCNCPoint4[20791] = {X 426.9642, Y 36.2780, Z -6.3333, A 0.000, B 0.000, C 0.000 }
gfCNCPoint4[20792] = {X 428.2756, Y 33.7112, Z -6.3333, A 0.000, B 0.000, C 0.000 }
gfCNCPoint4[20793] = {X 427.2117, Y 32.3941, Z -6.3333, A 0.000, B 0.000, C 0.000 }
gfCNCPoint4[20794] = {X 426.2869, Y 30.9760, Z -6.3333, A 0.000, B 0.000, C 0.000 }
gfCNCPoint4[20795] = {X 425.5106, Y 29.4714, Z -6.3333, A 0.000, B 0.000, C 0.000 }
gfCNCPoint4[20796] = {X 424.8909, Y 27.8959, Z -6.3333, A 0.000, B 0.000, C 0.000 }
gfCNCPoint4[20797] = {X 424.8186, Y 27.6757, Z -6.3333, A 0.000, B 0.000, C 0.000 }
gfCNCPoint4[20798] = {X 424.7493, Y 27.4544, Z -6.3333, A 0.000, B 0.000, C 0.000 }
gfCNCPoint4[20799] = {X 424.3068, Y 25.6987, Z -6.3333, A 0.000, B 0.000, C 0.000 }
gfCNCPoint4[20800] = {X 424.0108, Y 23.9124, Z -6.3333, A 0.000, B 0.000, C 0.000 }
gfCNCPoint4[20801] = {X 423.8634, Y 22.1078, Z -6.3333, A 0.000, B 0.000, C 0.000 }
gfCNCPoint4[20802] = {X 418.2389, Y 31.1545, Z -6.3333, A 0.000, B 0.000, C 0.000 }
gfCNCPoint4[20803] = {X 416.2007, Y 29.8873, Z -6.3333, A 0.000, B 0.000, C 0.000 }
gfCNCPoint4[20804] = {X 414.5076, Y 32.6105, Z -6.3333, A 0.000, B 0.000, C 0.000 }
gfCNCPoint4[20805] = {X 414.5081, Y 39.7465, Z -6.3333, A 0.000, B 0.000, C 0.000 }
gfCNCPoint4[20806] = {X 415.1568, Y 40.7518, Z -6.3333, A 0.000, B 0.000, C 0.000 }
gfCNCPoint4[20807] = {X 415.6349, Y 41.8484, Z -6.3333, A 0.000, B 0.000, C 0.000 }
gfCNCPoint4[20808] = {X 415.9301, Y 43.0077, Z -6.3333, A 0.000, B 0.000, C 0.000 }
gfCNCPoint4[20809] = {X 416.0347, Y 44.1995, Z -6.3333, A 0.000, B 0.000, C 0.000 }
gfCNCPoint4[20810] = {X 416.0347, Y 45.0000, Z -6.3333, A 0.000, B 0.000, C 0.000 }
gfCNCPoint4[20811] = {X 416.0201, Y 45.4609, Z -6.3333, A 0.000, B 0.000, C 0.000 }
gfCNCPoint4[20812] = {X 415.9763, Y 45.9200, Z -6.3333, A 0.000, B 0.000, C 0.000 }
gfCNCPoint4[20813] = {X 419.4886, Y 45.9200, Z -6.3333, A 0.000, B 0.000, C 0.000 }
gfCNCPoint4[20814] = {X 420.8957, Y 46.0022, Z -6.3333, A 0.000, B 0.000, C 0.000 }
gfCNCPoint4[20815] = {X 422.2836, Y 46.2478, Z -6.3333, A 0.000, B 0.000, C 0.000 }
gfCNCPoint4[20816] = {X 423.4822, Y 46.5992, Z -6.3333, A 0.000, B 0.000, C 0.000 }
gfCNCPoint4[20817] = {X 424.6380, Y 47.0725, Z -6.3333, A 0.000, B 0.000, C 0.000 }
gfCNCPoint4[20818] = {X 425.7388, Y 47.6626, Z -6.3333, A 0.000, B 0.000, C 0.000 }
gfCNCPoint4[20819] = {X 425.4600, Y 46.7984, Z -6.3333, A 0.000, B 0.000, C 0.000 }
gfCNCPoint4[20820] = {X 425.2910, Y 45.9063, Z -6.3333, A 0.000, B 0.000, C 0.000 }
gfCNCPoint4[20821] = {X 425.2344, Y 45.0000, Z -6.3333, A 0.000, B 0.000, C 0.000 }
gfCNCPoint4[20822] = {X 425.2344, Y 44.2089, Z -6.3333, A 0.000, B 0.000, C 0.000 }
gfCNCPoint4[20823] = {X 425.2353, Y 44.0976, Z -6.3333, A 0.000, B 0.000, C 0.000 }
gfCNCPoint4[20824] = {X 425.2378, Y 43.9863, Z -6.3333, A 0.000, B 0.000, C 0.000 }
gfCNCPoint4[20825] = {X 425.3770, Y 42.7748, Z -6.3333, A 0.000, B 0.000, C 0.000 }
gfCNCPoint4[20826] = {X 425.7165, Y 41.6036, Z -6.3333, A 0.000, B 0.000, C 0.000 }
gfCNCPoint4[20827] = {X 426.2468, Y 40.5054, Z -6.3333, A 0.000, B 0.000, C 0.000 }
gfCNCPoint4[20828] = {X 426.9528, Y 39.5112, Z -6.3333, A 0.000, B 0.000, C 0.000 }
gfCNCPoint4[20829] = {X 427.8150, Y 38.6488, Z -6.3333, A 0.000, B 0.000, C 0.000 }
gfCNCPoint4[20830] = {X 428.8090, Y 37.9424, Z -6.3333, A 0.000, B 0.000, C 0.000 }
gfCNCPoint4[20831] = {X 431.2063, Y 33.2499, Z -6.3333, A 0.000, B 0.000, C 0.000 }
gfCNCPoint4[20832] = {X 430.0998, Y 32.1506, Z -6.3333, A 0.000, B 0.000, C 0.000 }
gfCNCPoint4[20833] = {X 429.1199, Y 30.9372, Z -6.3333, A 0.000, B 0.000, C 0.000 }
gfCNCPoint4[20834] = {X 428.2781, Y 29.6241, Z -6.3333, A 0.000, B 0.000, C 0.000 }
gfCNCPoint4[20835] = {X 427.5846, Y 28.2271, Z -6.3333, A 0.000, B 0.000, C 0.000 }
gfCNCPoint4[20836] = {X 427.0476, Y 26.7628, Z -6.3333, A 0.000, B 0.000, C 0.000 }
gfCNCPoint4[20837] = {X 426.6550, Y 25.2024, Z -6.3333, A 0.000, B 0.000, C 0.000 }
gfCNCPoint4[20838] = {X 426.3923, Y 23.6150, Z -6.3333, A 0.000, B 0.000, C 0.000 }
gfCNCPoint4[20839] = {X 426.2614, Y 22.0113, Z -6.3333, A 0.000, B 0.000, C 0.000 }
gfCNCPoint4[20840] = {X 426.2916, Y 19.8883, Z -6.3333, A 0.000, B 0.000, C 0.000 }
gfCNCPoint4[20841] = {X 426.5524, Y 17.7812, Z -6.3333, A 0.000, B 0.000, C 0.000 }
gfCNCPoint4[20842] = {X 427.0407, Y 15.7149, Z -6.3333, A 0.000, B 0.000, C 0.000 }
gfCNCPoint4[20843] = {X 427.6623, Y 14.0043, Z -6.3333, A 0.000, B 0.000, C 0.000 }
gfCNCPoint4[20844] = {X 428.4893, Y 12.3830, Z -6.3333, A 0.000, B 0.000, C 0.000 }
gfCNCPoint4[20845] = {X 429.5091, Y 10.8756, Z -6.3333, A 0.000, B 0.000, C 0.000 }
gfCNCPoint4[20846] = {X 430.7064, Y 9.5049, Z -6.3333, A 0.000, B 0.000, C 0.000 }
gfCNCPoint4[20847] = {X 426.0925, Y 9.5049, Z -6.3333, A 0.000, B 0.000, C 0.000 }
gfCNCPoint4[20848] = {X 426.3754, Y 10.3750, Z -6.3333, A 0.000, B 0.000, C 0.000 }
gfCNCPoint4[20849] = {X 426.5470, Y 11.2737, Z -6.3333, A 0.000, B 0.000, C 0.000 }
gfCNCPoint4[20850] = {X 426.6045, Y 12.1868, Z -6.3333, A 0.000, B 0.000, C 0.000 }
gfCNCPoint4[20851] = {X 426.6044, Y 12.9915, Z -6.3333, A 0.000, B 0.000, C 0.000 }
gfCNCPoint4[20852] = {X 426.4808, Y 14.2923, Z -6.3333, A 0.000, B 0.000, C 0.000 }
gfCNCPoint4[20853] = {X 426.1285, Y 15.5507, Z -6.3333, A 0.000, B 0.000, C 0.000 }
gfCNCPoint4[20854] = {X 425.5588, Y 16.7266, Z -6.3333, A 0.000, B 0.000, C 0.000 }
gfCNCPoint4[20855] = {X 424.7896, Y 17.7829, Z -6.3333, A 0.000, B 0.000, C 0.000 }
gfCNCPoint4[20856] = {X 423.8453, Y 18.6862, Z -6.3333, A 0.000, B 0.000, C 0.000 }
gfCNCPoint4[20857] = {X 422.7558, Y 19.4077, Z -6.3333, A 0.000, B 0.000, C 0.000 }
gfCNCPoint4[20858] = {X 422.3660, Y 19.9718, Z -6.3333, A 0.000, B 0.000, C 0.000 }
gfCNCPoint4[20859] = {X 422.0035, Y 20.5538, Z -6.3333, A 0.000, B 0.000, C 0.000 }
gfCNCPoint4[20860] = {X 416.2007, Y 29.8873, Z -6.3333, A 0.000, B 0.000, C 0.000 }
gfCNCPoint4[20861] = {X 414.1625, Y 28.6201, Z -6.3333, A 0.000, B 0.000, C 0.000 }
gfCNCPoint4[20862] = {X 412.1076, Y 31.9254, Z -6.3333, A 0.000, B 0.000, C 0.000 }
gfCNCPoint4[20863] = {X 412.1082, Y 40.6515, Z -6.3333, A 0.000, B 0.000, C 0.000 }
gfCNCPoint4[20864] = {X 412.7499, Y 41.4081, Z -6.3333, A 0.000, B 0.000, C 0.000 }
gfCNCPoint4[20865] = {X 413.2297, Y 42.2765, Z -6.3333, A 0.000, B 0.000, C 0.000 }
gfCNCPoint4[20866] = {X 413.5285, Y 43.2225, Z -6.3333, A 0.000, B 0.000, C 0.000 }
gfCNCPoint4[20867] = {X 413.6347, Y 44.2089, Z -6.3333, A 0.000, B 0.000, C 0.000 }
gfCNCPoint4[20868] = {X 413.6347, Y 45.0000, Z -6.3333, A 0.000, B 0.000, C 0.000 }
gfCNCPoint4[20869] = {X 413.6249, Y 45.3090, Z -6.3333, A 0.000, B 0.000, C 0.000 }
gfCNCPoint4[20870] = {X 413.5956, Y 45.6167, Z -6.3333, A 0.000, B 0.000, C 0.000 }
gfCNCPoint4[20871] = {X 413.3652, Y 46.5992, Z -6.3333, A 0.000, B 0.000, C 0.000 }
gfCNCPoint4[20872] = {X 412.9377, Y 47.5134, Z -6.3333, A 0.000, B 0.000, C 0.000 }
gfCNCPoint4[20873] = {X 412.3313, Y 48.3200, Z -6.3333, A 0.000, B 0.000, C 0.000 }
gfCNCPoint4[20874] = {X 411.9795, Y 47.9934, Z -6.3333, A 0.000, B 0.000, C 0.000 }
gfCNCPoint4[20875] = {X 411.3003, Y 48.5889, Z -6.3333, A 0.000, B 0.000, C 0.000 }
gfCNCPoint4[20876] = {X 410.5138, Y 49.0331, Z -6.3333, A 0.000, B 0.000, C 0.000 }
gfCNCPoint4[20877] = {X 409.6532, Y 49.3073, Z -6.3333, A 0.000, B 0.000, C 0.000 }
gfCNCPoint4[20878] = {X 408.7547, Y 49.4000, Z -6.3333, A 0.000, B 0.000, C 0.000 }
gfCNCPoint4[20879] = {X 402.3112, Y 49.4000, Z -6.3333, A 0.000, B 0.000, C 0.000 }
gfCNCPoint4[20880] = {X 401.3321, Y 49.2897, Z -6.3333, A 0.000, B 0.000, C 0.000 }
gfCNCPoint4[20881] = {X 400.4021, Y 48.9643, Z -6.3333, A 0.000, B 0.000, C 0.000 }
gfCNCPoint4[20882] = {X 399.5678, Y 48.4400, Z -6.3333, A 0.000, B 0.000, C 0.000 }
gfCNCPoint4[20883] = {X 398.8711, Y 47.7433, Z -6.3333, A 0.000, B 0.000, C 0.000 }
gfCNCPoint4[20884] = {X 398.3469, Y 46.9091, Z -6.3333, A 0.000, B 0.000, C 0.000 }
gfCNCPoint4[20885] = {X 398.0215, Y 45.9791, Z -6.3333, A 0.000, B 0.000, C 0.000 }
gfCNCPoint4[20886] = {X 397.9112, Y 45.0000, Z -6.3333, A 0.000, B 0.000, C 0.000 }
gfCNCPoint4[20887] = {X 397.9116, Y 44.1518, Z -6.3333, A 0.000, B 0.000, C 0.000 }
gfCNCPoint4[20888] = {X 398.0215, Y 43.2300, Z -6.3333, A 0.000, B 0.000, C 0.000 }
gfCNCPoint4[20889] = {X 398.3223, Y 42.3519, Z -6.3333, A 0.000, B 0.000, C 0.000 }
gfCNCPoint4[20890] = {X 398.8006, Y 41.5563, Z -6.3333, A 0.000, B 0.000, C 0.000 }
gfCNCPoint4[20891] = {X 399.4352, Y 40.8789, Z -6.3333, A 0.000, B 0.000, C 0.000 }
gfCNCPoint4[20892] = {X 399.4352, Y 31.6966, Z -6.3333, A 0.000, B 0.000, C 0.000 }
gfCNCPoint4[20893] = {X 393.4509, Y 21.2900, Z -6.3333, A 0.000, B 0.000, C 0.000 }
gfCNCPoint4[20894] = {X 392.5630, Y 19.7793, Z -6.3333, A 0.000, B 0.000, C 0.000 }
gfCNCPoint4[20895] = {X 391.6466, Y 18.2859, Z -6.3333, A 0.000, B 0.000, C 0.000 }
gfCNCPoint4[20896] = {X 391.1738, Y 17.6274, Z -6.3333, A 0.000, B 0.000, C 0.000 }
gfCNCPoint4[20897] = {X 390.6224, Y 17.0333, Z -6.3333, A 0.000, B 0.000, C 0.000 }
gfCNCPoint4[20898] = {X 389.8675, Y 16.6247, Z -6.3333, A 0.000, B 0.000, C 0.000 }
gfCNCPoint4[20899] = {X 389.2064, Y 16.0773, Z -6.3333, A 0.000, B 0.000, C 0.000 }
gfCNCPoint4[20900] = {X 388.6641, Y 15.4119, Z -6.3333, A 0.000, B 0.000, C 0.000 }
gfCNCPoint4[20901] = {X 388.2613, Y 14.6540, Z -6.3333, A 0.000, B 0.000, C 0.000 }
gfCNCPoint4[20902] = {X 388.0133, Y 13.8322, Z -6.3333, A 0.000, B 0.000, C 0.000 }
gfCNCPoint4[20903] = {X 387.9296, Y 12.9780, Z -6.3333, A 0.000, B 0.000, C 0.000 }
gfCNCPoint4[20904] = {X 387.9296, Y 12.1868, Z -6.3333, A 0.000, B 0.000, C 0.000 }
gfCNCPoint4[20905] = {X 388.0399, Y 11.2077, Z -6.3333, A 0.000, B 0.000, C 0.000 }
gfCNCPoint4[20906] = {X 388.3654, Y 10.2777, Z -6.3333, A 0.000, B 0.000, C 0.000 }
gfCNCPoint4[20907] = {X 388.8896, Y 9.4435, Z -6.3333, A 0.000, B 0.000, C 0.000 }
gfCNCPoint4[20908] = {X 389.5863, Y 8.7468, Z -6.3333, A 0.000, B 0.000, C 0.000 }
gfCNCPoint4[20909] = {X 390.4205, Y 8.2226, Z -6.3333, A 0.000, B 0.000, C 0.000 }
gfCNCPoint4[20910] = {X 391.3505, Y 7.8971, Z -6.3333, A 0.000, B 0.000, C 0.000 }
gfCNCPoint4[20911] = {X 392.3296, Y 7.7868, Z -6.3333, A 0.000, B 0.000, C 0.000 }
gfCNCPoint4[20912] = {X 399.1118, Y 7.7868, Z -6.3333, A 0.000, B 0.000, C 0.000 }
gfCNCPoint4[20913] = {X 400.0909, Y 7.8971, Z -6.3333, A 0.000, B 0.000, C 0.000 }
gfCNCPoint4[20914] = {X 401.0208, Y 8.2226, Z -6.3333, A 0.000, B 0.000, C 0.000 }
gfCNCPoint4[20915] = {X 401.8551, Y 8.7468, Z -6.3333, A 0.000, B 0.000, C 0.000 }
gfCNCPoint4[20916] = {X 402.5518, Y 9.4435, Z -6.3333, A 0.000, B 0.000, C 0.000 }
gfCNCPoint4[20917] = {X 403.0760, Y 10.2777, Z -6.3333, A 0.000, B 0.000, C 0.000 }
gfCNCPoint4[20918] = {X 403.4014, Y 11.2077, Z -6.3333, A 0.000, B 0.000, C 0.000 }
gfCNCPoint4[20919] = {X 403.5118, Y 12.1868, Z -6.3333, A 0.000, B 0.000, C 0.000 }
gfCNCPoint4[20920] = {X 403.5115, Y 13.0233, Z -6.3333, A 0.000, B 0.000, C 0.000 }
gfCNCPoint4[20921] = {X 403.4070, Y 13.9326, Z -6.3333, A 0.000, B 0.000, C 0.000 }
gfCNCPoint4[20922] = {X 403.1165, Y 14.8007, Z -6.3333, A 0.000, B 0.000, C 0.000 }
gfCNCPoint4[20923] = {X 405.3501, Y 18.6790, Z -6.3333, A 0.000, B 0.000, C 0.000 }
gfCNCPoint4[20924] = {X 407.7807, Y 14.7421, Z -6.3333, A 0.000, B 0.000, C 0.000 }
gfCNCPoint4[20925] = {X 407.5048, Y 13.8791, Z -6.3333, A 0.000, B 0.000, C 0.000 }
gfCNCPoint4[20926] = {X 407.4115, Y 12.9780, Z -6.3333, A 0.000, B 0.000, C 0.000 }
gfCNCPoint4[20927] = {X 407.4115, Y 12.1868, Z -6.3333, A 0.000, B 0.000, C 0.000 }
gfCNCPoint4[20928] = {X 407.5219, Y 11.2077, Z -6.3333, A 0.000, B 0.000, C 0.000 }
gfCNCPoint4[20929] = {X 407.8473, Y 10.2777, Z -6.3333, A 0.000, B 0.000, C 0.000 }
gfCNCPoint4[20930] = {X 408.3715, Y 9.4435, Z -6.3333, A 0.000, B 0.000, C 0.000 }
gfCNCPoint4[20931] = {X 409.0682, Y 8.7468, Z -6.3333, A 0.000, B 0.000, C 0.000 }
gfCNCPoint4[20932] = {X 409.9025, Y 8.2226, Z -6.3333, A 0.000, B 0.000, C 0.000 }
gfCNCPoint4[20933] = {X 410.8324, Y 7.8971, Z -6.3333, A 0.000, B 0.000, C 0.000 }
gfCNCPoint4[20934] = {X 411.8115, Y 7.7868, Z -6.3333, A 0.000, B 0.000, C 0.000 }
gfCNCPoint4[20935] = {X 419.3245, Y 7.7868, Z -6.3333, A 0.000, B 0.000, C 0.000 }
gfCNCPoint4[20936] = {X 420.3036, Y 7.8971, Z -6.3333, A 0.000, B 0.000, C 0.000 }
gfCNCPoint4[20937] = {X 421.2335, Y 8.2226, Z -6.3333, A 0.000, B 0.000, C 0.000 }
gfCNCPoint4[20938] = {X 422.0678, Y 8.7468, Z -6.3333, A 0.000, B 0.000, C 0.000 }
gfCNCPoint4[20939] = {X 422.7645, Y 9.4435, Z -6.3333, A 0.000, B 0.000, C 0.000 }
gfCNCPoint4[20940] = {X 423.2887, Y 10.2777, Z -6.3333, A 0.000, B 0.000, C 0.000 }
gfCNCPoint4[20941] = {X 423.6141, Y 11.2077, Z -6.3333, A 0.000, B 0.000, C 0.000 }
gfCNCPoint4[20942] = {X 423.7245, Y 12.1868, Z -6.3333, A 0.000, B 0.000, C 0.000 }
gfCNCPoint4[20943] = {X 423.7245, Y 12.9807, Z -6.3333, A 0.000, B 0.000, C 0.000 }
gfCNCPoint4[20944] = {X 423.6309, Y 13.8596, Z -6.3333, A 0.000, B 0.000, C 0.000 }
gfCNCPoint4[20945] = {X 423.3659, Y 14.7028, Z -6.3333, A 0.000, B 0.000, C 0.000 }
gfCNCPoint4[20946] = {X 422.9400, Y 15.4772, Z -6.3333, A 0.000, B 0.000, C 0.000 }
gfCNCPoint4[20947] = {X 422.3697, Y 16.1524, Z -6.3333, A 0.000, B 0.000, C 0.000 }
gfCNCPoint4[20948] = {X 421.6775, Y 16.7020, Z -6.3333, A 0.000, B 0.000, C 0.000 }
gfCNCPoint4[20949] = {X 420.8906, Y 17.1043, Z -6.3333, A 0.000, B 0.000, C 0.000 }
gfCNCPoint4[20950] = {X 420.1835, Y 18.0570, Z -6.3333, A 0.000, B 0.000, C 0.000 }
gfCNCPoint4[20951] = {X 419.5435, Y 19.0559, Z -6.3333, A 0.000, B 0.000, C 0.000 }
gfCNCPoint4[20952] = {X 418.0618, Y 21.4545, Z -6.3333, A 0.000, B 0.000, C 0.000 }
gfCNCPoint4[20953] = {X 411.6276, Y 31.7882, Z -6.3333, A 0.000, B 0.000, C 0.000 }
gfCNCPoint4[20954] = {X 411.6282, Y 40.8614, Z -6.3333, A 0.000, B 0.000, C 0.000 }
gfCNCPoint4[20955] = {X 412.2673, Y 41.5582, Z -6.3333, A 0.000, B 0.000, C 0.000 }
gfCNCPoint4[20956] = {X 412.7475, Y 42.3728, Z -6.3333, A 0.000, B 0.000, C 0.000 }
gfCNCPoint4[20957] = {X 413.0476, Y 43.2694, Z -6.3333, A 0.000, B 0.000, C 0.000 }
gfCNCPoint4[20958] = {X 413.1547, Y 44.2089, Z -6.3333, A 0.000, B 0.000, C 0.000 }
gfCNCPoint4[20959] = {X 413.1545, Y 45.0423, Z -6.3333, A 0.000, B 0.000, C 0.000 }
gfCNCPoint4[20960] = {X 413.0719, Y 45.8494, Z -6.3333, A 0.000, B 0.000, C 0.000 }
gfCNCPoint4[20961] = {X 412.8426, Y 46.6276, Z -6.3333, A 0.000, B 0.000, C 0.000 }
gfCNCPoint4[20962] = {X 412.4743, Y 47.3505, Z -6.3333, A 0.000, B 0.000, C 0.000 }
gfCNCPoint4[20963] = {X 411.9795, Y 47.9934, Z -6.3333, A 0.000, B 0.000, C 0.000 }
gfCNCPoint4[20964] = {X 412.3313, Y 48.3200, Z -6.3333, A 0.000, B 0.000, C 0.000 }
gfCNCPoint4[20965] = {X 419.4886, Y 48.3200, Z -6.3333, A 0.000, B 0.000, C 0.000 }
gfCNCPoint4[20966] = {X 420.8006, Y 48.4093, Z -6.3333, A 0.000, B 0.000, C 0.000 }
gfCNCPoint4[20967] = {X 422.0883, Y 48.6756, Z -6.3333, A 0.000, B 0.000, C 0.000 }
gfCNCPoint4[20968] = {X 423.3281, Y 49.1140, Z -6.3333, A 0.000, B 0.000, C 0.000 }
gfCNCPoint4[20969] = {X 424.4970, Y 49.7164, Z -6.3333, A 0.000, B 0.000, C 0.000 }
gfCNCPoint4[20970] = {X 425.4625, Y 50.3832, Z -6.3333, A 0.000, B 0.000, C 0.000 }
gfCNCPoint4[20971] = {X 426.3402, Y 51.1620, Z -6.3333, A 0.000, B 0.000, C 0.000 }
gfCNCPoint4[20972] = {X 427.1172, Y 52.0412, Z -6.3333, A 0.000, B 0.000, C 0.000 }
gfCNCPoint4[20973] = {X 427.7821, Y 53.0080, Z -6.3333, A 0.000, B 0.000, C 0.000 }
gfCNCPoint4[20974] = {X 428.1266, Y 53.6310, Z -6.3333, A 0.000, B 0.000, C 0.000 }
gfCNCPoint4[20975] = {X 428.4243, Y 54.2776, Z -6.3333, A 0.000, B 0.000, C 0.000 }
gfCNCPoint4[20976] = {X 431.5823, Y 55.5081, Z -6.3333, A 0.000, B 0.000, C 0.000 }
gfCNCPoint4[20977] = {X 439.8791, Y 58.8000, Z -6.3333, A 0.000, B 0.000, C 0.000 }
gfCNCPoint4[20978] = {X 441.6493, Y 54.3384, Z -6.3333, A 0.000, B 0.000, C 0.000 }
gfCNCPoint4[20979] = {X 444.2224, Y 55.3593, Z -6.3333, A 0.000, B 0.000, C 0.000 }
gfCNCPoint4[20980] = {X 444.5427, Y 54.0014, Z -6.3333, A 0.000, B 0.000, C 0.000 }
gfCNCPoint4[20981] = {X 444.9921, Y 52.6806, Z -6.3333, A 0.000, B 0.000, C 0.000 }
gfCNCPoint4[20982] = {X 443.9526, Y 53.3761, Z -6.3333, A 0.000, B 0.000, C 0.000 }
gfCNCPoint4[20983] = {X 442.8321, Y 53.9318, Z -6.3333, A 0.000, B 0.000, C 0.000 }
gfCNCPoint4[20984] = {X 441.6493, Y 54.3384, Z -6.3333, A 0.000, B 0.000, C 0.000 }
gfCNCPoint4[20985] = {X 440.7642, Y 56.5692, Z -6.3333, A 0.000, B 0.000, C 0.000 }
gfCNCPoint4[20986] = {X 446.3797, Y 58.7973, Z -6.3333, A 0.000, B 0.000, C 0.000 }
gfCNCPoint4[20987] = {X 446.3796, Y 58.0000, Z -6.3333, A 0.000, B 0.000, C 0.000 }
gfCNCPoint4[20988] = {X 446.4304, Y 56.8939, Z -6.3333, A 0.000, B 0.000, C 0.000 }
gfCNCPoint4[20989] = {X 446.5822, Y 55.7970, Z -6.3333, A 0.000, B 0.000, C 0.000 }
gfCNCPoint4[20990] = {X 446.8493, Y 54.6641, Z -6.3333, A 0.000, B 0.000, C 0.000 }
gfCNCPoint4[20991] = {X 447.2243, Y 53.5622, Z -6.3333, A 0.000, B 0.000, C 0.000 }
gfCNCPoint4[20992] = {X 447.8767, Y 52.1752, Z -6.3333, A 0.000, B 0.000, C 0.000 }
gfCNCPoint4[20993] = {X 448.6995, Y 50.8820, Z -6.3333, A 0.000, B 0.000, C 0.000 }
gfCNCPoint4[20994] = {X 447.8224, Y 50.1272, Z -6.3333, A 0.000, B 0.000, C 0.000 }
gfCNCPoint4[20995] = {X 447.0760, Y 49.2431, Z -6.3333, A 0.000, B 0.000, C 0.000 }
gfCNCPoint4[20996] = {X 446.4792, Y 48.2518, Z -6.3333, A 0.000, B 0.000, C 0.000 }
gfCNCPoint4[20997] = {X 446.0469, Y 47.1785, Z -6.3333, A 0.000, B 0.000, C 0.000 }
gfCNCPoint4[20998] = {X 445.6333, Y 48.2126, Z -6.3333, A 0.000, B 0.000, C 0.000 }
gfCNCPoint4[20999] = {X 445.0668, Y 49.1715, Z -6.3333, A 0.000, B 0.000, C 0.000 }
gfCNCPoint4[21000] = {X 444.3606, Y 50.0328, Z -6.3333, A 0.000, B 0.000, C 0.000 }
gfCNCPoint4[21001] = {X 443.5314, Y 50.7763, Z -6.3333, A 0.000, B 0.000, C 0.000 }
gfCNCPoint4[21002] = {X 442.7496, Y 51.2994, Z -6.3333, A 0.000, B 0.000, C 0.000 }
gfCNCPoint4[21003] = {X 441.9069, Y 51.7173, Z -6.3333, A 0.000, B 0.000, C 0.000 }
gfCNCPoint4[21004] = {X 441.0174, Y 52.0231, Z -6.3333, A 0.000, B 0.000, C 0.000 }
gfCNCPoint4[21005] = {X 440.0675, Y 52.2155, Z -6.3333, A 0.000, B 0.000, C 0.000 }
gfCNCPoint4[21006] = {X 439.1005, Y 52.2800, Z -6.3333, A 0.000, B 0.000, C 0.000 }
gfCNCPoint4[21007] = {X 432.5144, Y 52.2800, Z -6.3333, A 0.000, B 0.000, C 0.000 }
gfCNCPoint4[21008] = {X 431.6034, Y 52.2228, Z -6.3333, A 0.000, B 0.000, C 0.000 }
gfCNCPoint4[21009] = {X 430.7066, Y 52.0520, Z -6.3333, A 0.000, B 0.000, C 0.000 }
gfCNCPoint4[21010] = {X 429.8384, Y 51.7703, Z -6.3333, A 0.000, B 0.000, C 0.000 }
gfCNCPoint4[21011] = {X 430.0167, Y 52.0768, Z -6.3333, A 0.000, B 0.000, C 0.000 }
gfCNCPoint4[21012] = {X 430.1861, Y 52.3883, Z -6.3333, A 0.000, B 0.000, C 0.000 }
gfCNCPoint4[21013] = {X 432.4640, Y 53.2759, Z -6.3333, A 0.000, B 0.000, C 0.000 }
gfCNCPoint4[21014] = {X 440.7642, Y 56.5692, Z -6.3333, A 0.000, B 0.000, C 0.000 }
gfCNCPoint4[21015] = {X 439.8791, Y 58.8000, Z -6.3333, A 0.000, B 0.000, C 0.000 }
gfCNCPoint4[21016] = {X 449.5092, Y 62.6210, Z -6.3333, A 0.000, B 0.000, C 0.000 }
gfCNCPoint4[21017] = {X 449.1113, Y 61.4462, Z -6.3333, A 0.000, B 0.000, C 0.000 }
gfCNCPoint4[21018] = {X 448.8668, Y 60.2303, Z -6.3333, A 0.000, B 0.000, C 0.000 }
gfCNCPoint4[21019] = {X 448.7798, Y 58.9930, Z -6.3333, A 0.000, B 0.000, C 0.000 }
gfCNCPoint4[21020] = {X 448.7796, Y 58.0000, Z -6.3333, A 0.000, B 0.000, C 0.000 }
gfCNCPoint4[21021] = {X 448.8564, Y 56.7833, Z -6.3333, A 0.000, B 0.000, C 0.000 }
gfCNCPoint4[21022] = {X 449.0855, Y 55.5859, Z -6.3333, A 0.000, B 0.000, C 0.000 }
gfCNCPoint4[21023] = {X 449.4632, Y 54.4268, Z -6.3333, A 0.000, B 0.000, C 0.000 }
gfCNCPoint4[21024] = {X 449.9837, Y 53.3244, Z -6.3333, A 0.000, B 0.000, C 0.000 }
gfCNCPoint4[21025] = {X 450.6386, Y 52.2961, Z -6.3333, A 0.000, B 0.000, C 0.000 }
gfCNCPoint4[21026] = {X 451.3887, Y 51.3890, Z -6.3333, A 0.000, B 0.000, C 0.000 }
gfCNCPoint4[21027] = {X 452.2434, Y 50.5796, Z -6.3333, A 0.000, B 0.000, C 0.000 }
gfCNCPoint4[21028] = {X 453.1901, Y 49.8800, Z -6.3333, A 0.000, B 0.000, C 0.000 }
gfCNCPoint4[21029] = {X 452.3731, Y 49.8442, Z -6.3333, A 0.000, B 0.000, C 0.000 }
gfCNCPoint4[21030] = {X 451.5735, Y 49.6724, Z -6.3333, A 0.000, B 0.000, C 0.000 }
gfCNCPoint4[21031] = {X 450.8138, Y 49.3696, Z -6.3333, A 0.000, B 0.000, C 0.000 }
gfCNCPoint4[21032] = {X 450.1154, Y 48.9441, Z -6.3333, A 0.000, B 0.000, C 0.000 }
gfCNCPoint4[21033] = {X 449.3503, Y 48.2496, Z -6.3333, A 0.000, B 0.000, C 0.000 }
gfCNCPoint4[21034] = {X 448.7486, Y 47.4095, Z -6.3333, A 0.000, B 0.000, C 0.000 }
gfCNCPoint4[21035] = {X 448.3373, Y 46.4616, Z -6.3333, A 0.000, B 0.000, C 0.000 }
gfCNCPoint4[21036] = {X 448.1732, Y 45.7588, Z -6.3333, A 0.000, B 0.000, C 0.000 }
gfCNCPoint4[21037] = {X 448.1146, Y 45.0395, Z -6.3333, A 0.000, B 0.000, C 0.000 }
gfCNCPoint4[21038] = {X 448.1149, Y 44.1417, Z -6.3333, A 0.000, B 0.000, C 0.000 }
gfCNCPoint4[21039] = {X 448.2252, Y 43.1751, Z -6.3333, A 0.000, B 0.000, C 0.000 }
gfCNCPoint4[21040] = {X 448.5250, Y 42.2497, Z -6.3333, A 0.000, B 0.000, C 0.000 }
gfCNCPoint4[21041] = {X 449.0024, Y 41.4021, Z -6.3333, A 0.000, B 0.000, C 0.000 }
gfCNCPoint4[21042] = {X 449.6384, Y 40.6660, Z -6.3333, A 0.000, B 0.000, C 0.000 }
gfCNCPoint4[21043] = {X 449.6384, Y 35.0338, Z -6.3333, A 0.000, B 0.000, C 0.000 }
gfCNCPoint4[21044] = {X 447.8172, Y 35.0338, Z -6.3333, A 0.000, B 0.000, C 0.000 }
gfCNCPoint4[21045] = {X 443.7930, Y 42.8691, Z -6.3333, A 0.000, B 0.000, C 0.000 }
gfCNCPoint4[21046] = {X 443.9303, Y 43.5109, Z -6.3333, A 0.000, B 0.000, C 0.000 }
gfCNCPoint4[21047] = {X 443.9803, Y 44.1653, Z -6.3333, A 0.000, B 0.000, C 0.000 }
gfCNCPoint4[21048] = {X 443.9805, Y 45.0000, Z -6.3333, A 0.000, B 0.000, C 0.000 }
gfCNCPoint4[21049] = {X 443.9242, Y 45.7387, Z -6.3333, A 0.000, B 0.000, C 0.000 }
gfCNCPoint4[21050] = {X 443.7568, Y 46.4603, Z -6.3333, A 0.000, B 0.000, C 0.000 }
gfCNCPoint4[21051] = {X 443.3474, Y 47.4038, Z -6.3333, A 0.000, B 0.000, C 0.000 }
gfCNCPoint4[21052] = {X 442.7493, Y 48.2405, Z -6.3333, A 0.000, B 0.000, C 0.000 }
gfCNCPoint4[21053] = {X 441.9891, Y 48.9332, Z -6.3333, A 0.000, B 0.000, C 0.000 }
gfCNCPoint4[21054] = {X 441.1006, Y 49.4513, Z -6.3333, A 0.000, B 0.000, C 0.000 }
gfCNCPoint4[21055] = {X 440.1232, Y 49.7716, Z -6.3333, A 0.000, B 0.000, C 0.000 }
gfCNCPoint4[21056] = {X 439.1005, Y 49.8800, Z -6.3333, A 0.000, B 0.000, C 0.000 }
gfCNCPoint4[21057] = {X 432.5144, Y 49.8800, Z -6.3333, A 0.000, B 0.000, C 0.000 }
gfCNCPoint4[21058] = {X 431.6014, Y 49.7938, Z -6.3333, A 0.000, B 0.000, C 0.000 }
gfCNCPoint4[21059] = {X 430.7206, Y 49.5383, Z -6.3333, A 0.000, B 0.000, C 0.000 }
gfCNCPoint4[21060] = {X 429.8343, Y 49.0782, Z -6.3333, A 0.000, B 0.000, C 0.000 }
gfCNCPoint4[21061] = {X 429.0603, Y 48.4473, Z -6.3333, A 0.000, B 0.000, C 0.000 }
gfCNCPoint4[21062] = {X 428.4309, Y 47.6720, Z -6.3333, A 0.000, B 0.000, C 0.000 }
gfCNCPoint4[21063] = {X 427.9725, Y 46.7848, Z -6.3333, A 0.000, B 0.000, C 0.000 }
gfCNCPoint4[21064] = {X 427.7197, Y 45.9083, Z -6.3333, A 0.000, B 0.000, C 0.000 }
gfCNCPoint4[21065] = {X 427.6344, Y 45.0000, Z -6.3333, A 0.000, B 0.000, C 0.000 }
gfCNCPoint4[21066] = {X 427.6344, Y 44.2089, Z -6.3333, A 0.000, B 0.000, C 0.000 }
gfCNCPoint4[21067] = {X 427.7263, Y 43.2661, Z -6.3333, A 0.000, B 0.000, C 0.000 }
gfCNCPoint4[21068] = {X 427.9987, Y 42.3588, Z -6.3333, A 0.000, B 0.000, C 0.000 }
gfCNCPoint4[21069] = {X 428.4412, Y 41.5212, Z -6.3333, A 0.000, B 0.000, C 0.000 }
gfCNCPoint4[21070] = {X 429.0371, Y 40.7849, Z -6.3333, A 0.000, B 0.000, C 0.000 }
gfCNCPoint4[21071] = {X 429.7641, Y 40.1776, Z -6.3333, A 0.000, B 0.000, C 0.000 }
gfCNCPoint4[21072] = {X 430.5947, Y 39.7222, Z -6.3333, A 0.000, B 0.000, C 0.000 }
gfCNCPoint4[21073] = {X 434.2529, Y 32.5618, Z -6.3333, A 0.000, B 0.000, C 0.000 }
gfCNCPoint4[21074] = {X 432.9254, Y 31.5656, Z -6.3333, A 0.000, B 0.000, C 0.000 }
gfCNCPoint4[21075] = {X 431.7498, Y 30.3941, Z -6.3333, A 0.000, B 0.000, C 0.000 }
gfCNCPoint4[21076] = {X 430.7489, Y 29.0702, Z -6.3333, A 0.000, B 0.000, C 0.000 }
gfCNCPoint4[21077] = {X 429.9423, Y 27.6197, Z -6.3333, A 0.000, B 0.000, C 0.000 }
gfCNCPoint4[21078] = {X 429.3457, Y 26.0709, Z -6.3333, A 0.000, B 0.000, C 0.000 }
gfCNCPoint4[21079] = {X 428.8991, Y 24.1612, Z -6.3333, A 0.000, B 0.000, C 0.000 }
gfCNCPoint4[21080] = {X 428.6741, Y 22.2128, Z -6.3333, A 0.000, B 0.000, C 0.000 }
gfCNCPoint4[21081] = {X 428.6735, Y 20.2515, Z -6.3333, A 0.000, B 0.000, C 0.000 }
gfCNCPoint4[21082] = {X 428.8974, Y 18.3031, Z -6.3333, A 0.000, B 0.000, C 0.000 }
gfCNCPoint4[21083] = {X 429.3429, Y 16.3931, Z -6.3333, A 0.000, B 0.000, C 0.000 }
gfCNCPoint4[21084] = {X 429.8636, Y 14.9604, Z -6.3333, A 0.000, B 0.000, C 0.000 }
gfCNCPoint4[21085] = {X 430.5563, Y 13.6025, Z -6.3333, A 0.000, B 0.000, C 0.000 }
gfCNCPoint4[21086] = {X 431.4106, Y 12.3400, Z -6.3333, A 0.000, B 0.000, C 0.000 }
gfCNCPoint4[21087] = {X 432.4134, Y 11.1920, Z -6.3333, A 0.000, B 0.000, C 0.000 }
gfCNCPoint4[21088] = {X 433.5450, Y 10.1794, Z -6.3333, A 0.000, B 0.000, C 0.000 }
gfCNCPoint4[21089] = {X 434.7920, Y 9.3129, Z -6.3333, A 0.000, B 0.000, C 0.000 }
gfCNCPoint4[21090] = {X 436.1356, Y 8.6054, Z -6.3333, A 0.000, B 0.000, C 0.000 }
gfCNCPoint4[21091] = {X 437.5556, Y 8.0677, Z -6.3333, A 0.000, B 0.000, C 0.000 }
gfCNCPoint4[21092] = {X 439.0308, Y 7.7076, Z -6.3333, A 0.000, B 0.000, C 0.000 }
gfCNCPoint4[21093] = {X 441.1775, Y 7.4104, Z -6.3333, A 0.000, B 0.000, C 0.000 }
gfCNCPoint4[21094] = {X 443.3426, Y 7.3140, Z -6.3333, A 0.000, B 0.000, C 0.000 }
gfCNCPoint4[21095] = {X 459.4468, Y 7.3099, Z -6.3333, A 0.000, B 0.000, C 0.000 }
gfCNCPoint4[21096] = {X 460.4097, Y 7.4060, Z -6.3333, A 0.000, B 0.000, C 0.000 }
gfCNCPoint4[21097] = {X 461.3346, Y 7.6906, Z -6.3333, A 0.000, B 0.000, C 0.000 }
gfCNCPoint4[21098] = {X 462.1850, Y 8.1523, Z -6.3333, A 0.000, B 0.000, C 0.000 }
gfCNCPoint4[21099] = {X 462.9273, Y 8.7731, Z -6.3333, A 0.000, B 0.000, C 0.000 }
gfCNCPoint4[21100] = {X 463.5323, Y 9.5283, Z -6.3333, A 0.000, B 0.000, C 0.000 }
gfCNCPoint4[21101] = {X 463.9760, Y 10.3882, Z -6.3333, A 0.000, B 0.000, C 0.000 }
gfCNCPoint4[21102] = {X 464.2317, Y 11.2685, Z -6.3333, A 0.000, B 0.000, C 0.000 }
gfCNCPoint4[21103] = {X 464.3179, Y 12.1810, Z -6.3333, A 0.000, B 0.000, C 0.000 }
gfCNCPoint4[21104] = {X 464.3179, Y 12.9780, Z -6.3333, A 0.000, B 0.000, C 0.000 }
gfCNCPoint4[21105] = {X 464.2174, Y 13.9634, Z -6.3333, A 0.000, B 0.000, C 0.000 }
gfCNCPoint4[21106] = {X 463.9200, Y 14.9083, Z -6.3333, A 0.000, B 0.000, C 0.000 }
gfCNCPoint4[21107] = {X 463.4378, Y 15.7736, Z -6.3333, A 0.000, B 0.000, C 0.000 }
gfCNCPoint4[21108] = {X 462.7909, Y 16.5237, Z -6.3333, A 0.000, B 0.000, C 0.000 }
gfCNCPoint4[21109] = {X 462.7906, Y 16.7696, Z -6.3333, A 0.000, B 0.000, C 0.000 }
gfCNCPoint4[21110] = {X 462.7916, Y 40.6638, Z -6.3333, A 0.000, B 0.000, C 0.000 }
gfCNCPoint4[21111] = {X 463.4323, Y 41.4053, Z -6.3333, A 0.000, B 0.000, C 0.000 }
gfCNCPoint4[21112] = {X 463.9118, Y 42.2598, Z -6.3333, A 0.000, B 0.000, C 0.000 }
gfCNCPoint4[21113] = {X 464.2110, Y 43.1929, Z -6.3333, A 0.000, B 0.000, C 0.000 }
gfCNCPoint4[21114] = {X 464.3178, Y 44.1670, Z -6.3333, A 0.000, B 0.000, C 0.000 }
gfCNCPoint4[21115] = {X 464.3179, Y 45.0000, Z -6.3333, A 0.000, B 0.000, C 0.000 }
gfCNCPoint4[21116] = {X 464.3082, Y 45.3090, Z -6.3333, A 0.000, B 0.000, C 0.000 }
gfCNCPoint4[21117] = {X 464.2788, Y 45.6167, Z -6.3333, A 0.000, B 0.000, C 0.000 }
gfCNCPoint4[21118] = {X 464.0485, Y 46.5992, Z -6.3333, A 0.000, B 0.000, C 0.000 }
gfCNCPoint4[21119] = {X 463.6209, Y 47.5134, Z -6.3333, A 0.000, B 0.000, C 0.000 }
gfCNCPoint4[21120] = {X 463.0145, Y 48.3200, Z -6.3333, A 0.000, B 0.000, C 0.000 }
gfCNCPoint4[21121] = {X 462.6627, Y 47.9934, Z -6.3333, A 0.000, B 0.000, C 0.000 }
gfCNCPoint4[21122] = {X 461.9835, Y 48.5889, Z -6.3333, A 0.000, B 0.000, C 0.000 }
gfCNCPoint4[21123] = {X 461.1970, Y 49.0331, Z -6.3333, A 0.000, B 0.000, C 0.000 }
gfCNCPoint4[21124] = {X 460.3364, Y 49.3073, Z -6.3333, A 0.000, B 0.000, C 0.000 }
gfCNCPoint4[21125] = {X 459.4379, Y 49.4000, Z -6.3333, A 0.000, B 0.000, C 0.000 }
gfCNCPoint4[21126] = {X 452.9945, Y 49.4000, Z -6.3333, A 0.000, B 0.000, C 0.000 }
gfCNCPoint4[21127] = {X 452.0154, Y 49.2897, Z -6.3333, A 0.000, B 0.000, C 0.000 }
gfCNCPoint4[21128] = {X 451.0854, Y 48.9643, Z -6.3333, A 0.000, B 0.000, C 0.000 }
gfCNCPoint4[21129] = {X 450.2511, Y 48.4400, Z -6.3333, A 0.000, B 0.000, C 0.000 }
gfCNCPoint4[21130] = {X 449.5544, Y 47.7433, Z -6.3333, A 0.000, B 0.000, C 0.000 }
gfCNCPoint4[21131] = {X 449.0302, Y 46.9091, Z -6.3333, A 0.000, B 0.000, C 0.000 }
gfCNCPoint4[21132] = {X 448.7048, Y 45.9791, Z -6.3333, A 0.000, B 0.000, C 0.000 }
gfCNCPoint4[21133] = {X 448.5945, Y 45.0000, Z -6.3333, A 0.000, B 0.000, C 0.000 }
gfCNCPoint4[21134] = {X 448.5949, Y 44.1483, Z -6.3333, A 0.000, B 0.000, C 0.000 }
gfCNCPoint4[21135] = {X 448.7053, Y 43.2275, Z -6.3333, A 0.000, B 0.000, C 0.000 }
gfCNCPoint4[21136] = {X 449.0063, Y 42.3503, Z -6.3333, A 0.000, B 0.000, C 0.000 }
gfCNCPoint4[21137] = {X 449.4844, Y 41.5556, Z -6.3333, A 0.000, B 0.000, C 0.000 }
gfCNCPoint4[21138] = {X 450.1184, Y 40.8789, Z -6.3333, A 0.000, B 0.000, C 0.000 }
gfCNCPoint4[21139] = {X 450.1184, Y 34.5538, Z -6.3333, A 0.000, B 0.000, C 0.000 }
gfCNCPoint4[21140] = {X 447.5241, Y 34.5538, Z -6.3333, A 0.000, B 0.000, C 0.000 }
gfCNCPoint4[21141] = {X 443.2767, Y 42.8236, Z -6.3333, A 0.000, B 0.000, C 0.000 }
gfCNCPoint4[21142] = {X 443.4442, Y 43.5073, Z -6.3333, A 0.000, B 0.000, C 0.000 }
gfCNCPoint4[21143] = {X 443.5005, Y 44.2089, Z -6.3333, A 0.000, B 0.000, C 0.000 }
gfCNCPoint4[21144] = {X 443.5005, Y 45.0000, Z -6.3333, A 0.000, B 0.000, C 0.000 }
gfCNCPoint4[21145] = {X 443.3902, Y 45.9791, Z -6.3333, A 0.000, B 0.000, C 0.000 }
gfCNCPoint4[21146] = {X 443.0647, Y 46.9091, Z -6.3333, A 0.000, B 0.000, C 0.000 }
gfCNCPoint4[21147] = {X 442.5405, Y 47.7434, Z -6.3333, A 0.000, B 0.000, C 0.000 }
gfCNCPoint4[21148] = {X 441.8438, Y 48.4401, Z -6.3333, A 0.000, B 0.000, C 0.000 }
gfCNCPoint4[21149] = {X 441.0096, Y 48.9643, Z -6.3333, A 0.000, B 0.000, C 0.000 }
gfCNCPoint4[21150] = {X 440.0796, Y 49.2897, Z -6.3333, A 0.000, B 0.000, C 0.000 }
gfCNCPoint4[21151] = {X 439.1005, Y 49.4000, Z -6.3333, A 0.000, B 0.000, C 0.000 }
gfCNCPoint4[21152] = {X 432.5144, Y 49.4000, Z -6.3333, A 0.000, B 0.000, C 0.000 }
gfCNCPoint4[21153] = {X 431.5353, Y 49.2897, Z -6.3333, A 0.000, B 0.000, C 0.000 }
gfCNCPoint4[21154] = {X 430.6053, Y 48.9643, Z -6.3333, A 0.000, B 0.000, C 0.000 }
gfCNCPoint4[21155] = {X 429.7711, Y 48.4401, Z -6.3333, A 0.000, B 0.000, C 0.000 }
gfCNCPoint4[21156] = {X 429.0743, Y 47.7434, Z -6.3333, A 0.000, B 0.000, C 0.000 }
gfCNCPoint4[21157] = {X 428.5501, Y 46.9091, Z -6.3333, A 0.000, B 0.000, C 0.000 }
gfCNCPoint4[21158] = {X 428.2247, Y 45.9791, Z -6.3333, A 0.000, B 0.000, C 0.000 }
gfCNCPoint4[21159] = {X 428.1144, Y 45.0000, Z -6.3333, A 0.000, B 0.000, C 0.000 }
gfCNCPoint4[21160] = {X 428.1148, Y 44.1483, Z -6.3333, A 0.000, B 0.000, C 0.000 }
gfCNCPoint4[21161] = {X 428.2132, Y 43.2816, Z -6.3333, A 0.000, B 0.000, C 0.000 }
gfCNCPoint4[21162] = {X 428.4806, Y 42.4514, Z -6.3333, A 0.000, B 0.000, C 0.000 }
gfCNCPoint4[21163] = {X 428.9065, Y 41.6903, Z -6.3333, A 0.000, B 0.000, C 0.000 }
gfCNCPoint4[21164] = {X 429.4741, Y 41.0281, Z -6.3333, A 0.000, B 0.000, C 0.000 }
gfCNCPoint4[21165] = {X 430.1613, Y 40.4909, Z -6.3333, A 0.000, B 0.000, C 0.000 }
gfCNCPoint4[21166] = {X 430.9408, Y 40.0998, Z -6.3333, A 0.000, B 0.000, C 0.000 }
gfCNCPoint4[21167] = {X 434.8813, Y 32.3868, Z -6.3333, A 0.000, B 0.000, C 0.000 }
gfCNCPoint4[21168] = {X 433.7236, Y 31.5991, Z -6.3333, A 0.000, B 0.000, C 0.000 }
gfCNCPoint4[21169] = {X 432.6711, Y 30.6755, Z -6.3333, A 0.000, B 0.000, C 0.000 }
gfCNCPoint4[21170] = {X 431.7399, Y 29.6298, Z -6.3333, A 0.000, B 0.000, C 0.000 }
gfCNCPoint4[21171] = {X 430.9438, Y 28.4778, Z -6.3333, A 0.000, B 0.000, C 0.000 }
gfCNCPoint4[21172] = {X 430.2950, Y 27.2369, Z -6.3333, A 0.000, B 0.000, C 0.000 }
gfCNCPoint4[21173] = {X 429.8033, Y 25.9258, Z -6.3333, A 0.000, B 0.000, C 0.000 }
gfCNCPoint4[21174] = {X 429.3707, Y 24.0712, Z -6.3333, A 0.000, B 0.000, C 0.000 }
gfCNCPoint4[21175] = {X 429.1529, Y 22.1794, Z -6.3333, A 0.000, B 0.000, C 0.000 }
gfCNCPoint4[21176] = {X 429.1529, Y 20.2751, Z -6.3333, A 0.000, B 0.000, C 0.000 }
gfCNCPoint4[21177] = {X 429.3707, Y 18.3832, Z -6.3333, A 0.000, B 0.000, C 0.000 }
gfCNCPoint4[21178] = {X 429.8033, Y 16.5287, Z -6.3333, A 0.000, B 0.000, C 0.000 }
gfCNCPoint4[21179] = {X 430.3769, Y 14.9871, Z -6.3333, A 0.000, B 0.000, C 0.000 }
gfCNCPoint4[21180] = {X 431.1574, Y 13.5393, Z -6.3333, A 0.000, B 0.000, C 0.000 }
gfCNCPoint4[21181] = {X 432.1299, Y 12.2128, Z -6.3333, A 0.000, B 0.000, C 0.000 }
gfCNCPoint4[21182] = {X 433.2760, Y 11.0330, Z -6.3333, A 0.000, B 0.000, C 0.000 }
gfCNCPoint4[21183] = {X 434.5736, Y 10.0223, Z -6.3333, A 0.000, B 0.000, C 0.000 }
gfCNCPoint4[21184] = {X 435.9982, Y 9.2001, Z -6.3333, A 0.000, B 0.000, C 0.000 }
gfCNCPoint4[21185] = {X 437.5224, Y 8.5820, Z -6.3333, A 0.000, B 0.000, C 0.000 }
gfCNCPoint4[21186] = {X 439.1173, Y 8.1798, Z -6.3333, A 0.000, B 0.000, C 0.000 }
gfCNCPoint4[21187] = {X 441.2214, Y 7.8884, Z -6.3333, A 0.000, B 0.000, C 0.000 }
gfCNCPoint4[21188] = {X 443.3434, Y 7.7940, Z -6.3333, A 0.000, B 0.000, C 0.000 }
gfCNCPoint4[21189] = {X 444.0367, Y 7.7899, Z -6.3333, A 0.000, B 0.000, C 0.000 }
gfCNCPoint4[21190] = {X 459.4468, Y 7.7899, Z -6.3333, A 0.000, B 0.000, C 0.000 }
gfCNCPoint4[21191] = {X 460.4239, Y 7.9000, Z -6.3333, A 0.000, B 0.000, C 0.000 }
gfCNCPoint4[21192] = {X 461.3521, Y 8.2248, Z -6.3333, A 0.000, B 0.000, C 0.000 }
gfCNCPoint4[21193] = {X 462.1846, Y 8.7479, Z -6.3333, A 0.000, B 0.000, C 0.000 }
gfCNCPoint4[21194] = {X 462.8799, Y 9.4432, Z -6.3333, A 0.000, B 0.000, C 0.000 }
gfCNCPoint4[21195] = {X 463.4031, Y 10.2758, Z -6.3333, A 0.000, B 0.000, C 0.000 }
gfCNCPoint4[21196] = {X 463.7278, Y 11.2039, Z -6.3333, A 0.000, B 0.000, C 0.000 }
gfCNCPoint4[21197] = {X 463.8379, Y 12.1810, Z -6.3333, A 0.000, B 0.000, C 0.000 }
gfCNCPoint4[21198] = {X 463.8377, Y 13.0201, Z -6.3333, A 0.000, B 0.000, C 0.000 }
gfCNCPoint4[21199] = {X 463.7300, Y 13.9468, Z -6.3333, A 0.000, B 0.000, C 0.000 }
gfCNCPoint4[21200] = {X 463.4292, Y 14.8299, Z -6.3333, A 0.000, B 0.000, C 0.000 }
gfCNCPoint4[21201] = {X 462.9491, Y 15.6298, Z -6.3333, A 0.000, B 0.000, C 0.000 }
gfCNCPoint4[21202] = {X 462.3111, Y 16.3104, Z -6.3333, A 0.000, B 0.000, C 0.000 }
gfCNCPoint4[21203] = {X 462.3106, Y 16.7691, Z -6.3333, A 0.000, B 0.000, C 0.000 }
gfCNCPoint4[21204] = {X 462.3116, Y 40.8769, Z -6.3333, A 0.000, B 0.000, C 0.000 }
gfCNCPoint4[21205] = {X 462.9558, Y 41.5659, Z -6.3333, A 0.000, B 0.000, C 0.000 }
gfCNCPoint4[21206] = {X 463.4382, Y 42.3764, Z -6.3333, A 0.000, B 0.000, C 0.000 }
gfCNCPoint4[21207] = {X 463.7369, Y 43.2711, Z -6.3333, A 0.000, B 0.000, C 0.000 }
gfCNCPoint4[21208] = {X 463.8379, Y 44.2088, Z -6.3333, A 0.000, B 0.000, C 0.000 }
gfCNCPoint4[21209] = {X 463.8379, Y 45.0000, Z -6.3333, A 0.000, B 0.000, C 0.000 }
gfCNCPoint4[21210] = {X 463.7612, Y 45.8182, Z -6.3333, A 0.000, B 0.000, C 0.000 }
gfCNCPoint4[21211] = {X 463.5336, Y 46.6079, Z -6.3333, A 0.000, B 0.000, C 0.000 }
gfCNCPoint4[21212] = {X 463.1632, Y 47.3415, Z -6.3333, A 0.000, B 0.000, C 0.000 }
gfCNCPoint4[21213] = {X 462.6627, Y 47.9934, Z -6.3333, A 0.000, B 0.000, C 0.000 }
gfCNCPoint4[21214] = {X 463.0145, Y 48.3200, Z -6.3333, A 0.000, B 0.000, C 0.000 }
gfCNCPoint4[21215] = {X 472.1884, Y 48.3200, Z -6.3333, A 0.000, B 0.000, C 0.000 }
gfCNCPoint4[21216] = {X 471.5820, Y 47.5134, Z -6.3333, A 0.000, B 0.000, C 0.000 }
gfCNCPoint4[21217] = {X 471.1544, Y 46.5992, Z -6.3333, A 0.000, B 0.000, C 0.000 }
gfCNCPoint4[21218] = {X 470.9241, Y 45.6167, Z -6.3333, A 0.000, B 0.000, C 0.000 }
gfCNCPoint4[21219] = {X 470.8947, Y 45.3090, Z -6.3333, A 0.000, B 0.000, C 0.000 }
gfCNCPoint4[21220] = {X 470.8850, Y 45.0000, Z -6.3333, A 0.000, B 0.000, C 0.000 }
gfCNCPoint4[21221] = {X 470.8850, Y 44.2089, Z -6.3333, A 0.000, B 0.000, C 0.000 }
gfCNCPoint4[21222] = {X 470.9769, Y 43.2661, Z -6.3333, A 0.000, B 0.000, C 0.000 }
gfCNCPoint4[21223] = {X 471.2492, Y 42.3588, Z -6.3333, A 0.000, B 0.000, C 0.000 }
gfCNCPoint4[21224] = {X 471.6917, Y 41.5212, Z -6.3333, A 0.000, B 0.000, C 0.000 }
gfCNCPoint4[21225] = {X 472.2877, Y 40.7849, Z -6.3333, A 0.000, B 0.000, C 0.000 }
gfCNCPoint4[21226] = {X 473.0147, Y 40.1776, Z -6.3333, A 0.000, B 0.000, C 0.000 }
gfCNCPoint4[21227] = {X 473.8453, Y 39.7222, Z -6.3333, A 0.000, B 0.000, C 0.000 }
gfCNCPoint4[21228] = {X 477.5001, Y 32.5683, Z -6.3333, A 0.000, B 0.000, C 0.000 }
gfCNCPoint4[21229] = {X 476.2822, Y 31.6588, Z -6.3333, A 0.000, B 0.000, C 0.000 }
gfCNCPoint4[21230] = {X 475.1888, Y 30.6027, Z -6.3333, A 0.000, B 0.000, C 0.000 }
gfCNCPoint4[21231] = {X 474.2376, Y 29.4171, Z -6.3333, A 0.000, B 0.000, C 0.000 }
gfCNCPoint4[21232] = {X 473.4437, Y 28.1208, Z -6.3333, A 0.000, B 0.000, C 0.000 }
gfCNCPoint4[21233] = {X 472.8198, Y 26.7346, Z -6.3333, A 0.000, B 0.000, C 0.000 }
gfCNCPoint4[21234] = {X 472.3760, Y 25.2808, Z -6.3333, A 0.000, B 0.000, C 0.000 }
gfCNCPoint4[21235] = {X 472.0517, Y 23.5415, Z -6.3333, A 0.000, B 0.000, C 0.000 }
gfCNCPoint4[21236] = {X 471.9068, Y 21.7783, Z -6.3333, A 0.000, B 0.000, C 0.000 }
gfCNCPoint4[21237] = {X 471.9427, Y 20.0094, Z -6.3333, A 0.000, B 0.000, C 0.000 }
gfCNCPoint4[21238] = {X 472.1591, Y 18.2535, Z -6.3333, A 0.000, B 0.000, C 0.000 }
gfCNCPoint4[21239] = {X 472.5537, Y 16.5288, Z -6.3333, A 0.000, B 0.000, C 0.000 }
gfCNCPoint4[21240] = {X 473.0724, Y 15.0578, Z -6.3333, A 0.000, B 0.000, C 0.000 }
gfCNCPoint4[21241] = {X 473.7719, Y 13.6637, Z -6.3333, A 0.000, B 0.000, C 0.000 }
gfCNCPoint4[21242] = {X 474.6408, Y 12.3684, Z -6.3333, A 0.000, B 0.000, C 0.000 }
gfCNCPoint4[21243] = {X 475.6656, Y 11.1925, Z -6.3333, A 0.000, B 0.000, C 0.000 }
gfCNCPoint4[21244] = {X 476.7432, Y 10.2233, Z -6.3333, A 0.000, B 0.000, C 0.000 }
gfCNCPoint4[21245] = {X 477.9265, Y 9.3866, Z -6.3333, A 0.000, B 0.000, C 0.000 }
gfCNCPoint4[21246] = {X 479.1994, Y 8.6938, Z -6.3333, A 0.000, B 0.000, C 0.000 }
gfCNCPoint4[21247] = {X 480.5445, Y 8.1542, Z -6.3333, A 0.000, B 0.000, C 0.000 }
gfCNCPoint4[21248] = {X 481.9433, Y 7.7754, Z -6.3333, A 0.000, B 0.000, C 0.000 }
gfCNCPoint4[21249] = {X 484.0946, Y 7.4402, Z -6.3333, A 0.000, B 0.000, C 0.000 }
gfCNCPoint4[21250] = {X 486.2687, Y 7.3221, Z -6.3333, A 0.000, B 0.000, C 0.000 }
gfCNCPoint4[21251] = {X 486.9707, Y 7.3099, Z -6.3333, A 0.000, B 0.000, C 0.000 }
gfCNCPoint4[21252] = {X 502.2122, Y 7.3099, Z -6.3333, A 0.000, B 0.000, C 0.000 }
gfCNCPoint4[21253] = {X 502.7439, Y 7.3141, Z -6.3333, A 0.000, B 0.000, C 0.000 }
gfCNCPoint4[21254] = {X 503.6983, Y 7.4163, Z -6.3333, A 0.000, B 0.000, C 0.000 }
gfCNCPoint4[21255] = {X 504.6140, Y 7.7039, Z -6.3333, A 0.000, B 0.000, C 0.000 }
gfCNCPoint4[21256] = {X 505.4553, Y 8.1659, Z -6.3333, A 0.000, B 0.000, C 0.000 }
gfCNCPoint4[21257] = {X 506.1896, Y 8.7841, Z -6.3333, A 0.000, B 0.000, C 0.000 }
gfCNCPoint4[21258] = {X 506.7881, Y 9.5344, Z -6.3333, A 0.000, B 0.000, C 0.000 }
gfCNCPoint4[21259] = {X 507.2275, Y 10.3878, Z -6.3333, A 0.000, B 0.000, C 0.000 }
gfCNCPoint4[21260] = {X 507.4825, Y 11.2660, Z -6.3333, A 0.000, B 0.000, C 0.000 }
gfCNCPoint4[21261] = {X 507.5685, Y 12.1765, Z -6.3333, A 0.000, B 0.000, C 0.000 }
gfCNCPoint4[21262] = {X 507.5683, Y 13.0237, Z -6.3333, A 0.000, B 0.000, C 0.000 }
gfCNCPoint4[21263] = {X 507.4609, Y 13.9969, Z -6.3333, A 0.000, B 0.000, C 0.000 }
gfCNCPoint4[21264] = {X 507.1615, Y 14.9290, Z -6.3333, A 0.000, B 0.000, C 0.000 }
gfCNCPoint4[21265] = {X 506.6820, Y 15.7827, Z -6.3333, A 0.000, B 0.000, C 0.000 }
gfCNCPoint4[21266] = {X 506.0418, Y 16.5234, Z -6.3333, A 0.000, B 0.000, C 0.000 }
gfCNCPoint4[21267] = {X 506.0417, Y 40.6634, Z -6.3333, A 0.000, B 0.000, C 0.000 }
gfCNCPoint4[21268] = {X 506.6825, Y 41.4048, Z -6.3333, A 0.000, B 0.000, C 0.000 }
gfCNCPoint4[21269] = {X 507.1622, Y 42.2593, Z -6.3333, A 0.000, B 0.000, C 0.000 }
gfCNCPoint4[21270] = {X 507.4615, Y 43.1924, Z -6.3333, A 0.000, B 0.000, C 0.000 }
gfCNCPoint4[21271] = {X 507.5683, Y 44.1665, Z -6.3333, A 0.000, B 0.000, C 0.000 }
gfCNCPoint4[21272] = {X 507.5685, Y 45.0000, Z -6.3333, A 0.000, B 0.000, C 0.000 }
gfCNCPoint4[21273] = {X 507.4747, Y 45.9520, Z -6.3333, A 0.000, B 0.000, C 0.000 }
gfCNCPoint4[21274] = {X 507.1970, Y 46.8675, Z -6.3333, A 0.000, B 0.000, C 0.000 }
gfCNCPoint4[21275] = {X 506.7461, Y 47.7112, Z -6.3333, A 0.000, B 0.000, C 0.000 }
gfCNCPoint4[21276] = {X 506.1392, Y 48.4507, Z -6.3333, A 0.000, B 0.000, C 0.000 }
gfCNCPoint4[21277] = {X 505.3997, Y 49.0576, Z -6.3333, A 0.000, B 0.000, C 0.000 }
gfCNCPoint4[21278] = {X 504.5560, Y 49.5085, Z -6.3333, A 0.000, B 0.000, C 0.000 }
gfCNCPoint4[21279] = {X 503.6405, Y 49.7862, Z -6.3333, A 0.000, B 0.000, C 0.000 }
gfCNCPoint4[21280] = {X 502.6885, Y 49.8800, Z -6.3333, A 0.000, B 0.000, C 0.000 }
gfCNCPoint4[21281] = {X 496.2450, Y 49.8800, Z -6.3333, A 0.000, B 0.000, C 0.000 }
gfCNCPoint4[21282] = {X 495.2220, Y 49.7716, Z -6.3333, A 0.000, B 0.000, C 0.000 }
gfCNCPoint4[21283] = {X 494.2445, Y 49.4511, Z -6.3333, A 0.000, B 0.000, C 0.000 }
gfCNCPoint4[21284] = {X 493.3559, Y 48.9328, Z -6.3333, A 0.000, B 0.000, C 0.000 }
gfCNCPoint4[21285] = {X 492.5956, Y 48.2398, Z -6.3333, A 0.000, B 0.000, C 0.000 }
gfCNCPoint4[21286] = {X 491.9976, Y 47.4028, Z -6.3333, A 0.000, B 0.000, C 0.000 }
gfCNCPoint4[21287] = {X 491.5882, Y 46.4590, Z -6.3333, A 0.000, B 0.000, C 0.000 }
gfCNCPoint4[21288] = {X 491.4241, Y 45.7570, Z -6.3333, A 0.000, B 0.000, C 0.000 }
gfCNCPoint4[21289] = {X 491.3652, Y 45.0385, Z -6.3333, A 0.000, B 0.000, C 0.000 }
gfCNCPoint4[21290] = {X 491.3655, Y 44.1416, Z -6.3333, A 0.000, B 0.000, C 0.000 }
gfCNCPoint4[21291] = {X 491.4758, Y 43.1751, Z -6.3333, A 0.000, B 0.000, C 0.000 }
gfCNCPoint4[21292] = {X 491.7756, Y 42.2496, Z -6.3333, A 0.000, B 0.000, C 0.000 }
gfCNCPoint4[21293] = {X 492.2530, Y 41.4020, Z -6.3333, A 0.000, B 0.000, C 0.000 }
gfCNCPoint4[21294] = {X 492.8890, Y 40.6660, Z -6.3333, A 0.000, B 0.000, C 0.000 }
gfCNCPoint4[21295] = {X 492.8890, Y 35.0338, Z -6.3333, A 0.000, B 0.000, C 0.000 }
gfCNCPoint4[21296] = {X 491.0670, Y 35.0338, Z -6.3333, A 0.000, B 0.000, C 0.000 }
gfCNCPoint4[21297] = {X 487.0435, Y 42.8691, Z -6.3333, A 0.000, B 0.000, C 0.000 }
gfCNCPoint4[21298] = {X 487.1808, Y 43.5106, Z -6.3333, A 0.000, B 0.000, C 0.000 }
gfCNCPoint4[21299] = {X 487.2308, Y 44.1648, Z -6.3333, A 0.000, B 0.000, C 0.000 }
gfCNCPoint4[21300] = {X 487.2310, Y 45.0000, Z -6.3333, A 0.000, B 0.000, C 0.000 }
gfCNCPoint4[21301] = {X 487.1749, Y 45.7380, Z -6.3333, A 0.000, B 0.000, C 0.000 }
gfCNCPoint4[21302] = {X 487.0078, Y 46.4590, Z -6.3333, A 0.000, B 0.000, C 0.000 }
gfCNCPoint4[21303] = {X 486.5939, Y 47.4110, Z -6.3333, A 0.000, B 0.000, C 0.000 }
gfCNCPoint4[21304] = {X 485.9879, Y 48.2538, Z -6.3333, A 0.000, B 0.000, C 0.000 }
gfCNCPoint4[21305] = {X 485.2175, Y 48.9494, Z -6.3333, A 0.000, B 0.000, C 0.000 }
gfCNCPoint4[21306] = {X 484.3173, Y 49.4663, Z -6.3333, A 0.000, B 0.000, C 0.000 }
gfCNCPoint4[21307] = {X 483.3557, Y 49.7755, Z -6.3333, A 0.000, B 0.000, C 0.000 }
gfCNCPoint4[21308] = {X 482.3510, Y 49.8800, Z -6.3333, A 0.000, B 0.000, C 0.000 }
gfCNCPoint4[21309] = {X 480.2695, Y 49.8800, Z -6.3333, A 0.000, B 0.000, C 0.000 }
gfCNCPoint4[21310] = {X 480.2695, Y 49.4000, Z -6.3333, A 0.000, B 0.000, C 0.000 }
gfCNCPoint4[21311] = {X 475.7650, Y 49.4000, Z -6.3333, A 0.000, B 0.000, C 0.000 }
gfCNCPoint4[21312] = {X 474.7859, Y 49.2897, Z -6.3333, A 0.000, B 0.000, C 0.000 }
gfCNCPoint4[21313] = {X 473.8559, Y 48.9643, Z -6.3333, A 0.000, B 0.000, C 0.000 }
gfCNCPoint4[21314] = {X 473.0216, Y 48.4401, Z -6.3333, A 0.000, B 0.000, C 0.000 }
gfCNCPoint4[21315] = {X 472.3249, Y 47.7434, Z -6.3333, A 0.000, B 0.000, C 0.000 }
gfCNCPoint4[21316] = {X 471.8007, Y 46.9091, Z -6.3333, A 0.000, B 0.000, C 0.000 }
gfCNCPoint4[21317] = {X 471.4753, Y 45.9791, Z -6.3333, A 0.000, B 0.000, C 0.000 }
gfCNCPoint4[21318] = {X 471.3650, Y 45.0000, Z -6.3333, A 0.000, B 0.000, C 0.000 }
gfCNCPoint4[21319] = {X 471.3654, Y 44.1483, Z -6.3333, A 0.000, B 0.000, C 0.000 }
gfCNCPoint4[21320] = {X 471.4638, Y 43.2816, Z -6.3333, A 0.000, B 0.000, C 0.000 }
gfCNCPoint4[21321] = {X 471.7311, Y 42.4514, Z -6.3333, A 0.000, B 0.000, C 0.000 }
gfCNCPoint4[21322] = {X 472.1570, Y 41.6903, Z -6.3333, A 0.000, B 0.000, C 0.000 }
gfCNCPoint4[21323] = {X 472.7247, Y 41.0281, Z -6.3333, A 0.000, B 0.000, C 0.000 }
gfCNCPoint4[21324] = {X 473.4118, Y 40.4909, Z -6.3333, A 0.000, B 0.000, C 0.000 }
gfCNCPoint4[21325] = {X 474.1914, Y 40.0998, Z -6.3333, A 0.000, B 0.000, C 0.000 }
gfCNCPoint4[21326] = {X 478.1276, Y 32.3951, Z -6.3333, A 0.000, B 0.000, C 0.000 }
gfCNCPoint4[21327] = {X 476.8702, Y 31.5214, Z -6.3333, A 0.000, B 0.000, C 0.000 }
gfCNCPoint4[21328] = {X 475.7396, Y 30.4890, Z -6.3333, A 0.000, B 0.000, C 0.000 }
gfCNCPoint4[21329] = {X 474.7557, Y 29.3159, Z -6.3333, A 0.000, B 0.000, C 0.000 }
gfCNCPoint4[21330] = {X 473.9358, Y 28.0227, Z -6.3333, A 0.000, B 0.000, C 0.000 }
gfCNCPoint4[21331] = {X 473.2945, Y 26.6324, Z -6.3333, A 0.000, B 0.000, C 0.000 }
gfCNCPoint4[21332] = {X 472.8429, Y 25.1694, Z -6.3333, A 0.000, B 0.000, C 0.000 }
gfCNCPoint4[21333] = {X 472.5275, Y 23.4783, Z -6.3333, A 0.000, B 0.000, C 0.000 }
gfCNCPoint4[21334] = {X 472.3865, Y 21.7638, Z -6.3333, A 0.000, B 0.000, C 0.000 }
gfCNCPoint4[21335] = {X 472.4214, Y 20.0439, Z -6.3333, A 0.000, B 0.000, C 0.000 }
gfCNCPoint4[21336] = {X 472.6318, Y 18.3366, Z -6.3333, A 0.000, B 0.000, C 0.000 }
gfCNCPoint4[21337] = {X 473.0155, Y 16.6597, Z -6.3333, A 0.000, B 0.000, C 0.000 }
gfCNCPoint4[21338] = {X 473.5621, Y 15.1345, Z -6.3333, A 0.000, B 0.000, C 0.000 }
gfCNCPoint4[21339] = {X 474.3106, Y 13.6975, Z -6.3333, A 0.000, B 0.000, C 0.000 }
gfCNCPoint4[21340] = {X 475.2471, Y 12.3754, Z -6.3333, A 0.000, B 0.000, C 0.000 }
gfCNCPoint4[21341] = {X 476.3544, Y 11.1926, Z -6.3333, A 0.000, B 0.000, C 0.000 }
gfCNCPoint4[21342] = {X 477.6119, Y 10.1710, Z -6.3333, A 0.000, B 0.000, C 0.000 }
gfCNCPoint4[21343] = {X 478.9964, Y 9.3294, Z -6.3333, A 0.000, B 0.000, C 0.000 }
gfCNCPoint4[21344] = {X 480.4822, Y 8.6835, Z -6.3333, A 0.000, B 0.000, C 0.000 }
gfCNCPoint4[21345] = {X 482.0420, Y 8.2451, Z -6.3333, A 0.000, B 0.000, C 0.000 }
gfCNCPoint4[21346] = {X 484.1468, Y 7.9174, Z -6.3333, A 0.000, B 0.000, C 0.000 }
gfCNCPoint4[21347] = {X 486.2739, Y 7.8021, Z -6.3333, A 0.000, B 0.000, C 0.000 }
gfCNCPoint4[21348] = {X 486.9707, Y 7.7899, Z -6.3333, A 0.000, B 0.000, C 0.000 }
gfCNCPoint4[21349] = {X 502.2084, Y 7.7899, Z -6.3333, A 0.000, B 0.000, C 0.000 }
gfCNCPoint4[21350] = {X 502.7401, Y 7.7941, Z -6.3333, A 0.000, B 0.000, C 0.000 }
gfCNCPoint4[21351] = {X 503.7097, Y 7.9104, Z -6.3333, A 0.000, B 0.000, C 0.000 }
gfCNCPoint4[21352] = {X 504.6294, Y 8.2386, Z -6.3333, A 0.000, B 0.000, C 0.000 }
gfCNCPoint4[21353] = {X 505.4537, Y 8.7623, Z -6.3333, A 0.000, B 0.000, C 0.000 }
gfCNCPoint4[21354] = {X 506.1415, Y 9.4555, Z -6.3333, A 0.000, B 0.000, C 0.000 }
gfCNCPoint4[21355] = {X 506.6587, Y 10.2838, Z -6.3333, A 0.000, B 0.000, C 0.000 }
gfCNCPoint4[21356] = {X 506.9797, Y 11.2061, Z -6.3333, A 0.000, B 0.000, C 0.000 }
gfCNCPoint4[21357] = {X 507.0885, Y 12.1765, Z -6.3333, A 0.000, B 0.000, C 0.000 }
gfCNCPoint4[21358] = {X 507.0883, Y 13.0233, Z -6.3333, A 0.000, B 0.000, C 0.000 }
gfCNCPoint4[21359] = {X 506.9800, Y 13.9491, Z -6.3333, A 0.000, B 0.000, C 0.000 }
gfCNCPoint4[21360] = {X 506.6792, Y 14.8313, Z -6.3333, A 0.000, B 0.000, C 0.000 }
gfCNCPoint4[21361] = {X 506.1993, Y 15.6303, Z -6.3333, A 0.000, B 0.000, C 0.000 }
gfCNCPoint4[21362] = {X 505.5618, Y 16.3103, Z -6.3333, A 0.000, B 0.000, C 0.000 }
gfCNCPoint4[21363] = {X 505.5617, Y 40.8765, Z -6.3333, A 0.000, B 0.000, C 0.000 }
gfCNCPoint4[21364] = {X 506.2060, Y 41.5655, Z -6.3333, A 0.000, B 0.000, C 0.000 }
gfCNCPoint4[21365] = {X 506.6887, Y 42.3761, Z -6.3333, A 0.000, B 0.000, C 0.000 }
gfCNCPoint4[21366] = {X 506.9874, Y 43.2709, Z -6.3333, A 0.000, B 0.000, C 0.000 }
gfCNCPoint4[21367] = {X 507.0885, Y 44.2089, Z -6.3333, A 0.000, B 0.000, C 0.000 }
gfCNCPoint4[21368] = {X 507.0885, Y 45.0000, Z -6.3333, A 0.000, B 0.000, C 0.000 }
gfCNCPoint4[21369] = {X 506.9782, Y 45.9791, Z -6.3333, A 0.000, B 0.000, C 0.000 }
gfCNCPoint4[21370] = {X 506.6528, Y 46.9091, Z -6.3333, A 0.000, B 0.000, C 0.000 }
gfCNCPoint4[21371] = {X 506.1285, Y 47.7434, Z -6.3333, A 0.000, B 0.000, C 0.000 }
gfCNCPoint4[21372] = {X 505.4318, Y 48.4401, Z -6.3333, A 0.000, B 0.000, C 0.000 }
gfCNCPoint4[21373] = {X 504.5976, Y 48.9643, Z -6.3333, A 0.000, B 0.000, C 0.000 }
gfCNCPoint4[21374] = {X 503.6676, Y 49.2897, Z -6.3333, A 0.000, B 0.000, C 0.000 }
gfCNCPoint4[21375] = {X 502.6885, Y 49.4000, Z -6.3333, A 0.000, B 0.000, C 0.000 }
gfCNCPoint4[21376] = {X 496.2450, Y 49.4000, Z -6.3333, A 0.000, B 0.000, C 0.000 }
gfCNCPoint4[21377] = {X 495.2659, Y 49.2897, Z -6.3333, A 0.000, B 0.000, C 0.000 }
gfCNCPoint4[21378] = {X 494.3359, Y 48.9643, Z -6.3333, A 0.000, B 0.000, C 0.000 }
gfCNCPoint4[21379] = {X 493.5017, Y 48.4400, Z -6.3333, A 0.000, B 0.000, C 0.000 }
gfCNCPoint4[21380] = {X 492.8050, Y 47.7433, Z -6.3333, A 0.000, B 0.000, C 0.000 }
gfCNCPoint4[21381] = {X 492.2808, Y 46.9091, Z -6.3333, A 0.000, B 0.000, C 0.000 }
gfCNCPoint4[21382] = {X 491.9553, Y 45.9791, Z -6.3333, A 0.000, B 0.000, C 0.000 }
gfCNCPoint4[21383] = {X 491.8450, Y 45.0000, Z -6.3333, A 0.000, B 0.000, C 0.000 }
gfCNCPoint4[21384] = {X 491.8454, Y 44.1483, Z -6.3333, A 0.000, B 0.000, C 0.000 }
gfCNCPoint4[21385] = {X 491.9559, Y 43.2275, Z -6.3333, A 0.000, B 0.000, C 0.000 }
gfCNCPoint4[21386] = {X 492.2568, Y 42.3503, Z -6.3333, A 0.000, B 0.000, C 0.000 }
gfCNCPoint4[21387] = {X 492.7349, Y 41.5556, Z -6.3333, A 0.000, B 0.000, C 0.000 }
gfCNCPoint4[21388] = {X 493.3690, Y 40.8789, Z -6.3333, A 0.000, B 0.000, C 0.000 }
gfCNCPoint4[21389] = {X 493.3690, Y 34.5538, Z -6.3333, A 0.000, B 0.000, C 0.000 }
gfCNCPoint4[21390] = {X 490.7739, Y 34.5538, Z -6.3333, A 0.000, B 0.000, C 0.000 }
gfCNCPoint4[21391] = {X 486.5273, Y 42.8236, Z -6.3333, A 0.000, B 0.000, C 0.000 }
gfCNCPoint4[21392] = {X 486.6947, Y 43.5073, Z -6.3333, A 0.000, B 0.000, C 0.000 }
gfCNCPoint4[21393] = {X 486.7510, Y 44.2089, Z -6.3333, A 0.000, B 0.000, C 0.000 }
gfCNCPoint4[21394] = {X 486.7510, Y 45.0000, Z -6.3333, A 0.000, B 0.000, C 0.000 }
gfCNCPoint4[21395] = {X 486.6407, Y 45.9791, Z -6.3333, A 0.000, B 0.000, C 0.000 }
gfCNCPoint4[21396] = {X 486.3153, Y 46.9091, Z -6.3333, A 0.000, B 0.000, C 0.000 }
gfCNCPoint4[21397] = {X 485.7911, Y 47.7434, Z -6.3333, A 0.000, B 0.000, C 0.000 }
gfCNCPoint4[21398] = {X 485.0944, Y 48.4401, Z -6.3333, A 0.000, B 0.000, C 0.000 }
gfCNCPoint4[21399] = {X 484.2601, Y 48.9643, Z -6.3333, A 0.000, B 0.000, C 0.000 }
gfCNCPoint4[21400] = {X 483.3301, Y 49.2897, Z -6.3333, A 0.000, B 0.000, C 0.000 }
gfCNCPoint4[21401] = {X 482.3510, Y 49.4000, Z -6.3333, A 0.000, B 0.000, C 0.000 }
gfCNCPoint4[21402] = {X 480.2695, Y 49.4000, Z -6.3333, A 0.000, B 0.000, C 0.000 }
gfCNCPoint4[21403] = {X 480.2695, Y 49.8800, Z -6.3333, A 0.000, B 0.000, C 0.000 }
gfCNCPoint4[21404] = {X 481.4067, Y 50.7435, Z -6.3333, A 0.000, B 0.000, C 0.000 }
gfCNCPoint4[21405] = {X 482.4044, Y 51.7649, Z -6.3333, A 0.000, B 0.000, C 0.000 }
gfCNCPoint4[21406] = {X 483.2411, Y 52.9219, Z -6.3333, A 0.000, B 0.000, C 0.000 }
gfCNCPoint4[21407] = {X 483.8615, Y 54.1044, Z -6.3333, A 0.000, B 0.000, C 0.000 }
gfCNCPoint4[21408] = {X 484.3133, Y 55.3610, Z -6.3333, A 0.000, B 0.000, C 0.000 }
gfCNCPoint4[21409] = {X 484.5879, Y 56.6678, Z -6.3333, A 0.000, B 0.000, C 0.000 }
gfCNCPoint4[21410] = {X 484.6800, Y 58.0000, Z -6.3333, A 0.000, B 0.000, C 0.000 }
gfCNCPoint4[21411] = {X 484.6797, Y 59.0140, Z -6.3333, A 0.000, B 0.000, C 0.000 }
gfCNCPoint4[21412] = {X 484.5592, Y 60.4583, Z -6.3333, A 0.000, B 0.000, C 0.000 }
gfCNCPoint4[21413] = {X 484.2245, Y 61.8684, Z -6.3333, A 0.000, B 0.000, C 0.000 }
gfCNCPoint4[21414] = {X 483.6831, Y 63.2127, Z -6.3333, A 0.000, B 0.000, C 0.000 }
gfCNCPoint4[21415] = {X 482.9469, Y 64.4611, Z -6.3333, A 0.000, B 0.000, C 0.000 }
gfCNCPoint4[21416] = {X 482.0327, Y 65.5857, Z -6.3333, A 0.000, B 0.000, C 0.000 }
gfCNCPoint4[21417] = {X 480.9608, Y 66.5611, Z -6.3333, A 0.000, B 0.000, C 0.000 }
gfCNCPoint4[21418] = {X 480.9611, Y 89.4453, Z -6.3333, A 0.000, B 0.000, C 0.000 }
gfCNCPoint4[21419] = {X 482.0601, Y 90.4476, Z -6.3333, A 0.000, B 0.000, C 0.000 }
gfCNCPoint4[21420] = {X 482.9921, Y 91.6067, Z -6.3333, A 0.000, B 0.000, C 0.000 }
gfCNCPoint4[21421] = {X 483.7351, Y 92.8951, Z -6.3333, A 0.000, B 0.000, C 0.000 }
gfCNCPoint4[21422] = {X 507.6813, Y 92.8951, Z -6.3333, A 0.000, B 0.000, C 0.000 }
gfCNCPoint4[21423] = {X 507.6813, Y 95.2951, Z -6.3333, A 0.000, B 0.000, C 0.000 }
gfCNCPoint4[21424] = {X 595.2966, Y 95.2951, Z -6.3333, A 0.000, B 0.000, C 0.000 }
gfCNCPoint4[21425] = {X 595.2966, Y 54.2000, Z -6.3333, A 0.000, B 0.000, C 0.000 }
gfCNCPoint4[21426] = {X 593.5565, Y 54.2000, Z -6.3333, A 0.000, B 0.000, C 0.000 }
gfCNCPoint4[21427] = {X 592.2403, Y 54.1053, Z -6.3333, A 0.000, B 0.000, C 0.000 }
gfCNCPoint4[21428] = {X 590.9511, Y 53.8233, Z -6.3333, A 0.000, B 0.000, C 0.000 }
gfCNCPoint4[21429] = {X 589.7155, Y 53.3598, Z -6.3333, A 0.000, B 0.000, C 0.000 }
gfCNCPoint4[21430] = {X 588.5589, Y 52.7242, Z -6.3333, A 0.000, B 0.000, C 0.000 }
gfCNCPoint4[21431] = {X 587.5052, Y 51.9297, Z -6.3333, A 0.000, B 0.000, C 0.000 }
gfCNCPoint4[21432] = {X 586.4956, Y 52.6955, Z -6.3333, A 0.000, B 0.000, C 0.000 }
gfCNCPoint4[21433] = {X 585.3903, Y 53.3153, Z -6.3333, A 0.000, B 0.000, C 0.000 }
gfCNCPoint4[21434] = {X 584.1375, Y 53.7999, Z -6.3333, A 0.000, B 0.000, C 0.000 }
gfCNCPoint4[21435] = {X 582.8276, Y 54.0969, Z -6.3333, A 0.000, B 0.000, C 0.000 }
gfCNCPoint4[21436] = {X 581.4884, Y 54.1999, Z -6.3333, A 0.000, B 0.000, C 0.000 }
gfCNCPoint4[21437] = {X 580.1485, Y 54.1069, Z -6.3333, A 0.000, B 0.000, C 0.000 }
gfCNCPoint4[21438] = {X 578.8364, Y 53.8198, Z -6.3333, A 0.000, B 0.000, C 0.000 }
gfCNCPoint4[21439] = {X 577.5801, Y 53.3447, Z -6.3333, A 0.000, B 0.000, C 0.000 }
gfCNCPoint4[21440] = {X 576.4063, Y 52.6917, Z -6.3333, A 0.000, B 0.000, C 0.000 }
gfCNCPoint4[21441] = {X 575.3401, Y 51.8748, Z -6.3333, A 0.000, B 0.000, C 0.000 }
gfCNCPoint4[21442] = {X 574.2798, Y 52.6879, Z -6.3333, A 0.000, B 0.000, C 0.000 }
gfCNCPoint4[21443] = {X 573.1128, Y 53.3388, Z -6.3333, A 0.000, B 0.000, C 0.000 }
gfCNCPoint4[21444] = {X 571.8638, Y 53.8139, Z -6.3333, A 0.000, B 0.000, C 0.000 }
gfCNCPoint4[21445] = {X 570.5592, Y 54.1030, Z -6.3333, A 0.000, B 0.000, C 0.000 }
gfCNCPoint4[21446] = {X 569.2264, Y 54.2000, Z -6.3333, A 0.000, B 0.000, C 0.000 }
gfCNCPoint4[21447] = {X 562.4443, Y 54.2000, Z -6.3333, A 0.000, B 0.000, C 0.000 }
gfCNCPoint4[21448] = {X 561.1326, Y 54.1060, Z -6.3333, A 0.000, B 0.000, C 0.000 }
gfCNCPoint4[21449] = {X 559.8478, Y 53.8260, Z -6.3333, A 0.000, B 0.000, C 0.000 }
gfCNCPoint4[21450] = {X 558.6160, Y 53.3656, Z -6.3333, A 0.000, B 0.000, C 0.000 }
gfCNCPoint4[21451] = {X 557.4624, Y 52.7344, Z -6.3333, A 0.000, B 0.000, C 0.000 }
gfCNCPoint4[21452] = {X 556.4106, Y 51.9451, Z -6.3333, A 0.000, B 0.000, C 0.000 }
gfCNCPoint4[21453] = {X 555.4849, Y 51.0172, Z -6.3333, A 0.000, B 0.000, C 0.000 }
gfCNCPoint4[21454] = {X 554.7005, Y 49.9672, Z -6.3333, A 0.000, B 0.000, C 0.000 }
gfCNCPoint4[21455] = {X 554.0732, Y 48.8164, Z -6.3333, A 0.000, B 0.000, C 0.000 }
gfCNCPoint4[21456] = {X 553.6158, Y 47.5881, Z -6.3333, A 0.000, B 0.000, C 0.000 }
gfCNCPoint4[21457] = {X 553.3377, Y 46.3073, Z -6.3333, A 0.000, B 0.000, C 0.000 }
gfCNCPoint4[21458] = {X 553.2443, Y 45.0000, Z -6.3333, A 0.000, B 0.000, C 0.000 }
gfCNCPoint4[21459] = {X 553.2443, Y 44.0472, Z -6.3333, A 0.000, B 0.000, C 0.000 }
gfCNCPoint4[21460] = {X 553.3460, Y 42.7142, Z -6.3333, A 0.000, B 0.000, C 0.000 }
gfCNCPoint4[21461] = {X 553.6391, Y 41.4099, Z -6.3333, A 0.000, B 0.000, C 0.000 }
gfCNCPoint4[21462] = {X 554.1175, Y 40.1616, Z -6.3333, A 0.000, B 0.000, C 0.000 }
gfCNCPoint4[21463] = {X 554.7712, Y 38.9954, Z -6.3333, A 0.000, B 0.000, C 0.000 }
gfCNCPoint4[21464] = {X 554.7712, Y 11.0098, Z -6.3333, A 0.000, B 0.000, C 0.000 }
gfCNCPoint4[21465] = {X 554.1214, Y 9.8545, Z -6.3333, A 0.000, B 0.000, C 0.000 }
gfCNCPoint4[21466] = {X 553.6445, Y 8.6179, Z -6.3333, A 0.000, B 0.000, C 0.000 }
gfCNCPoint4[21467] = {X 553.3501, Y 7.3255, Z -6.3333, A 0.000, B 0.000, C 0.000 }
gfCNCPoint4[21468] = {X 553.2446, Y 6.0043, Z -6.3333, A 0.000, B 0.000, C 0.000 }
gfCNCPoint4[21469] = {X 553.2443, Y 5.0000, Z -6.3333, A 0.000, B 0.000, C 0.000 }
gfCNCPoint4[21470] = {X 553.2455, Y 4.8524, Z -6.3333, A 0.000, B 0.000, C 0.000 }
gfCNCPoint4[21471] = {X 553.2490, Y 4.7049, Z -6.3333, A 0.000, B 0.000, C 0.000 }
gfCNCPoint4[21472] = {X 365.1879, Y 4.7049, Z -6.3333, A 0.000, B 0.000, C 0.000 }
gfCNCPoint4[21473] = {X 365.6160, Y 5.1721, Z -6.3333, A 0.000, B 0.000, C 0.000 }
gfCNCPoint4[21474] = {X 366.0315, Y 5.6504, Z -6.3333, A 0.000, B 0.000, C 0.000 }
gfCNCPoint4[21475] = {X 367.1004, Y 7.0011, Z -6.3333, A 0.000, B 0.000, C 0.000 }
gfCNCPoint4[21476] = {X 368.0843, Y 8.4148, Z -6.3333, A 0.000, B 0.000, C 0.000 }
gfCNCPoint4[21477] = {X 369.2517, Y 10.3771, Z -6.3333, A 0.000, B 0.000, C 0.000 }
gfCNCPoint4[21478] = {X 370.2556, Y 12.4279, Z -6.3333, A 0.000, B 0.000, C 0.000 }
gfCNCPoint4[21479] = {X 371.0895, Y 14.5534, Z -6.3333, A 0.000, B 0.000, C 0.000 }
gfCNCPoint4[21480] = {X 371.7478, Y 16.7397, Z -6.3333, A 0.000, B 0.000, C 0.000 }
gfCNCPoint4[21481] = {X 372.2263, Y 18.9723, Z -6.3333, A 0.000, B 0.000, C 0.000 }
gfCNCPoint4[21482] = {X 372.5872, Y 21.5596, Z -6.3333, A 0.000, B 0.000, C 0.000 }
gfCNCPoint4[21483] = {X 372.7524, Y 24.1667, Z -6.3333, A 0.000, B 0.000, C 0.000 }
gfCNCPoint4[21484] = {X 372.7212, Y 26.7788, Z -6.3333, A 0.000, B 0.000, C 0.000 }
gfCNCPoint4[21485] = {X 372.4935, Y 29.3812, Z -6.3333, A 0.000, B 0.000, C 0.000 }
gfCNCPoint4[21486] = {X 372.0707, Y 31.9591, Z -6.3333, A 0.000, B 0.000, C 0.000 }
gfCNCPoint4[21487] = {X 371.4844, Y 34.3140, Z -6.3333, A 0.000, B 0.000, C 0.000 }
gfCNCPoint4[21488] = {X 370.6926, Y 36.6081, Z -6.3333, A 0.000, B 0.000, C 0.000 }
gfCNCPoint4[21489] = {X 369.7017, Y 38.8233, Z -6.3333, A 0.000, B 0.000, C 0.000 }
gfCNCPoint4[21490] = {X 368.5192, Y 40.9426, Z -6.3333, A 0.000, B 0.000, C 0.000 }
gfCNCPoint4[21491] = {X 367.1545, Y 42.9493, Z -6.3333, A 0.000, B 0.000, C 0.000 }
gfCNCPoint4[21492] = {X 367.0390, Y 43.1073, Z -6.3333, A 0.000, B 0.000, C 0.000 }
gfCNCPoint4[21493] = {X 365.7258, Y 44.7100, Z -6.3333, A 0.000, B 0.000, C 0.000 }
gfCNCPoint4[21494] = {X 364.2842, Y 46.1981, Z -6.3333, A 0.000, B 0.000, C 0.000 }
gfCNCPoint4[21495] = {X 362.7241, Y 47.5615, Z -6.3333, A 0.000, B 0.000, C 0.000 }
gfCNCPoint4[21496] = {X 361.0563, Y 48.7907, Z -6.3333, A 0.000, B 0.000, C 0.000 }
gfCNCPoint4[21497] = {X 359.2921, Y 49.8772, Z -6.3333, A 0.000, B 0.000, C 0.000 }
gfCNCPoint4[21498] = {X 357.4439, Y 50.8136, Z -6.3333, A 0.000, B 0.000, C 0.000 }
gfCNCPoint4[21499] = {X 355.4662, Y 51.5793, Z -6.3333, A 0.000, B 0.000, C 0.000 }
gfCNCPoint4[21500] = {X 353.4326, Y 52.1813, Z -6.3333, A 0.000, B 0.000, C 0.000 }
gfCNCPoint4[21501] = {X 351.3567, Y 52.6153, Z -6.3333, A 0.000, B 0.000, C 0.000 }
gfCNCPoint4[21502] = {X 349.2523, Y 52.8787, Z -6.3333, A 0.000, B 0.000, C 0.000 }
gfCNCPoint4[21503] = {X 347.1334, Y 52.9695, Z -6.3333, A 0.000, B 0.000, C 0.000 }
gfCNCPoint4[21504] = {X 344.8131, Y 52.9272, Z -6.3333, A 0.000, B 0.000, C 0.000 }
gfCNCPoint4[21505] = {X 342.5051, Y 52.6840, Z -6.3333, A 0.000, B 0.000, C 0.000 }
gfCNCPoint4[21506] = {X 340.2269, Y 52.2419, Z -6.3333, A 0.000, B 0.000, C 0.000 }
gfCNCPoint4[21507] = {X 337.9955, Y 51.6041, Z -6.3333, A 0.000, B 0.000, C 0.000 }
gfCNCPoint4[21508] = {X 335.8278, Y 50.7754, Z -6.3333, A 0.000, B 0.000, C 0.000 }
gfCNCPoint4[21509] = {X 333.7400, Y 49.7621, Z -6.3333, A 0.000, B 0.000, C 0.000 }
gfCNCPoint4[21510] = {X 332.8348, Y 49.2288, Z -6.3333, A 0.000, B 0.000, C 0.000 }
gfCNCPoint4[21511] = {X 331.9511, Y 48.6605, Z -6.3333, A 0.000, B 0.000, C 0.000 }
gfCNCPoint4[21512] = {X 331.3041, Y 48.2123, Z -6.3333, A 0.000, B 0.000, C 0.000 }
gfCNCPoint4[21513] = {X 330.6704, Y 47.7454, Z -6.3333, A 0.000, B 0.000, C 0.000 }
gfCNCPoint4[21514] = {X 329.2186, Y 49.6564, Z -6.3333, A 0.000, B 0.000, C 0.000 }
gfCNCPoint4[21515] = {X 328.8734, Y 49.3901, Z -6.3333, A 0.000, B 0.000, C 0.000 }
gfCNCPoint4[21516] = {X 328.5322, Y 49.1187, Z -6.3333, A 0.000, B 0.000, C 0.000 }
gfCNCPoint4[21517] = {X 328.1269, Y 49.0391, Z -6.3333, A 0.000, B 0.000, C 0.000 }
gfCNCPoint4[21518] = {X 327.7253, Y 48.9423, Z -6.3333, A 0.000, B 0.000, C 0.000 }
gfCNCPoint4[21519] = {X 328.4872, Y 49.2674, Z -6.3333, A 0.000, B 0.000, C 0.000 }
gfCNCPoint4[21520] = {X 329.2186, Y 49.6564, Z -6.3333, A 0.000, B 0.000, C 0.000 }
gfCNCPoint4[21521] = {X 330.6704, Y 47.7454, Z -6.3333, A 0.000, B 0.000, C 0.000 }
gfCNCPoint4[21522] = {X 330.0961, Y 47.2966, Z -6.3333, A 0.000, B 0.000, C 0.000 }
gfCNCPoint4[21523] = {X 329.5341, Y 46.8324, Z -6.3333, A 0.000, B 0.000, C 0.000 }
gfCNCPoint4[21524] = {X 328.9314, Y 46.7520, Z -6.3333, A 0.000, B 0.000, C 0.000 }
gfCNCPoint4[21525] = {X 328.3374, Y 46.6216, Z -6.3333, A 0.000, B 0.000, C 0.000 }
gfCNCPoint4[21526] = {X 327.9789, Y 46.5172, Z -6.3333, A 0.000, B 0.000, C 0.000 }
gfCNCPoint4[21527] = {X 327.6263, Y 46.3944, Z -6.3333, A 0.000, B 0.000, C 0.000 }
gfCNCPoint4[21528] = {X 326.7320, Y 45.9864, Z -6.3333, A 0.000, B 0.000, C 0.000 }
gfCNCPoint4[21529] = {X 325.9009, Y 45.4616, Z -6.3333, A 0.000, B 0.000, C 0.000 }
gfCNCPoint4[21530] = {X 325.1480, Y 44.8296, Z -6.3333, A 0.000, B 0.000, C 0.000 }
gfCNCPoint4[21531] = {X 324.5140, Y 44.2115, Z -6.3333, A 0.000, B 0.000, C 0.000 }
gfCNCPoint4[21532] = {X 324.0475, Y 43.7117, Z -6.3333, A 0.000, B 0.000, C 0.000 }
gfCNCPoint4[21533] = {X 323.6300, Y 43.1703, Z -6.3333, A 0.000, B 0.000, C 0.000 }
gfCNCPoint4[21534] = {X 319.6957, Y 45.9200, Z -6.3333, A 0.000, B 0.000, C 0.000 }
gfCNCPoint4[21535] = {X 319.4780, Y 45.5976, Z -6.3333, A 0.000, B 0.000, C 0.000 }
gfCNCPoint4[21536] = {X 319.2708, Y 45.2683, Z -6.3333, A 0.000, B 0.000, C 0.000 }
gfCNCPoint4[21537] = {X 319.2514, Y 45.5948, Z -6.3333, A 0.000, B 0.000, C 0.000 }
gfCNCPoint4[21538] = {X 319.2174, Y 45.9200, Z -6.3333, A 0.000, B 0.000, C 0.000 }
gfCNCPoint4[21539] = {X 319.6957, Y 45.9200, Z -6.3333, A 0.000, B 0.000, C 0.000 }
gfCNCPoint4[21540] = {X 321.6628, Y 44.5452, Z -6.3333, A 0.000, B 0.000, C 0.000 }
gfCNCPoint4[21541] = {X 321.4884, Y 44.2868, Z -6.3333, A 0.000, B 0.000, C 0.000 }
gfCNCPoint4[21542] = {X 321.3224, Y 44.0230, Z -6.3333, A 0.000, B 0.000, C 0.000 }
gfCNCPoint4[21543] = {X 320.6709, Y 42.7448, Z -6.3333, A 0.000, B 0.000, C 0.000 }
gfCNCPoint4[21544] = {X 320.2154, Y 41.3843, Z -6.3333, A 0.000, B 0.000, C 0.000 }
gfCNCPoint4[21545] = {X 319.9660, Y 39.9715, Z -6.3333, A 0.000, B 0.000, C 0.000 }
gfCNCPoint4[21546] = {X 319.9282, Y 38.5373, Z -6.3333, A 0.000, B 0.000, C 0.000 }
gfCNCPoint4[21547] = {X 320.1028, Y 37.1133, Z -6.3333, A 0.000, B 0.000, C 0.000 }
gfCNCPoint4[21548] = {X 320.4309, Y 35.8883, Z -6.3333, A 0.000, B 0.000, C 0.000 }
gfCNCPoint4[21549] = {X 320.9164, Y 34.7167, Z -6.3333, A 0.000, B 0.000, C 0.000 }
gfCNCPoint4[21550] = {X 321.5508, Y 33.6186, Z -6.3333, A 0.000, B 0.000, C 0.000 }
gfCNCPoint4[21551] = {X 324.1389, Y 29.7495, Z -6.3333, A 0.000, B 0.000, C 0.000 }
gfCNCPoint4[21552] = {X 320.1492, Y 27.0808, Z -6.3333, A 0.000, B 0.000, C 0.000 }
gfCNCPoint4[21553] = {X 321.8650, Y 24.5157, Z -6.3333, A 0.000, B 0.000, C 0.000 }
gfCNCPoint4[21554] = {X 322.0211, Y 24.2912, Z -6.3333, A 0.000, B 0.000, C 0.000 }
gfCNCPoint4[21555] = {X 322.1814, Y 24.0697, Z -6.3333, A 0.000, B 0.000, C 0.000 }
gfCNCPoint4[21556] = {X 321.5380, Y 23.0772, Z -6.3333, A 0.000, B 0.000, C 0.000 }
gfCNCPoint4[21557] = {X 320.9777, Y 22.0354, Z -6.3333, A 0.000, B 0.000, C 0.000 }
gfCNCPoint4[21558] = {X 320.1494, Y 20.3315, Z -6.3333, A 0.000, B 0.000, C 0.000 }
gfCNCPoint4[21559] = {X 320.1492, Y 27.0808, Z -6.3333, A 0.000, B 0.000, C 0.000 }
gfCNCPoint4[21560] = {X 322.1440, Y 28.4152, Z -6.3333, A 0.000, B 0.000, C 0.000 }
gfCNCPoint4[21561] = {X 323.8536, Y 25.8595, Z -6.3333, A 0.000, B 0.000, C 0.000 }
gfCNCPoint4[21562] = {X 324.5431, Y 24.9455, Z -6.3333, A 0.000, B 0.000, C 0.000 }
gfCNCPoint4[21563] = {X 325.3162, Y 24.1010, Z -6.3333, A 0.000, B 0.000, C 0.000 }
gfCNCPoint4[21564] = {X 324.4812, Y 23.1413, Z -6.3333, A 0.000, B 0.000, C 0.000 }
gfCNCPoint4[21565] = {X 323.7518, Y 22.0990, Z -6.3333, A 0.000, B 0.000, C 0.000 }
gfCNCPoint4[21566] = {X 323.1360, Y 20.9859, Z -6.3333, A 0.000, B 0.000, C 0.000 }
gfCNCPoint4[21567] = {X 319.6151, Y 13.7428, Z -6.3333, A 0.000, B 0.000, C 0.000 }
gfCNCPoint4[21568] = {X 319.4387, Y 13.3633, Z -6.3333, A 0.000, B 0.000, C 0.000 }
gfCNCPoint4[21569] = {X 319.2755, Y 12.9779, Z -6.3333, A 0.000, B 0.000, C 0.000 }
gfCNCPoint4[21570] = {X 319.2755, Y 13.0353, Z -6.3333, A 0.000, B 0.000, C 0.000 }
gfCNCPoint4[21571] = {X 319.1698, Y 14.2151, Z -6.3333, A 0.000, B 0.000, C 0.000 }
gfCNCPoint4[21572] = {X 318.8743, Y 15.3621, Z -6.3333, A 0.000, B 0.000, C 0.000 }
gfCNCPoint4[21573] = {X 318.3966, Y 16.4460, Z -6.3333, A 0.000, B 0.000, C 0.000 }
gfCNCPoint4[21574] = {X 317.7495, Y 17.4381, Z -6.3333, A 0.000, B 0.000, C 0.000 }
gfCNCPoint4[21575] = {X 317.7488, Y 36.6455, Z -6.3333, A 0.000, B 0.000, C 0.000 }
gfCNCPoint4[21576] = {X 318.1583, Y 35.1168, Z -6.3333, A 0.000, B 0.000, C 0.000 }
gfCNCPoint4[21577] = {X 318.7641, Y 33.6548, Z -6.3333, A 0.000, B 0.000, C 0.000 }
gfCNCPoint4[21578] = {X 319.5559, Y 32.2844, Z -6.3333, A 0.000, B 0.000, C 0.000 }
gfCNCPoint4[21579] = {X 322.1440, Y 28.4152, Z -6.3333, A 0.000, B 0.000, C 0.000 }
gfCNCPoint4[21580] = {X 324.1389, Y 29.7495, Z -6.3333, A 0.000, B 0.000, C 0.000 }
gfCNCPoint4[21581] = {X 325.8357, Y 27.2126, Z -6.3333, A 0.000, B 0.000, C 0.000 }
gfCNCPoint4[21582] = {X 326.3883, Y 26.4803, Z -6.3333, A 0.000, B 0.000, C 0.000 }
gfCNCPoint4[21583] = {X 327.0077, Y 25.8035, Z -6.3333, A 0.000, B 0.000, C 0.000 }
gfCNCPoint4[21584] = {X 328.0707, Y 24.8904, Z -6.3333, A 0.000, B 0.000, C 0.000 }
gfCNCPoint4[21585] = {X 329.2543, Y 24.1403, Z -6.3333, A 0.000, B 0.000, C 0.000 }
gfCNCPoint4[21586] = {X 328.0859, Y 23.3667, Z -6.3333, A 0.000, B 0.000, C 0.000 }
gfCNCPoint4[21587] = {X 327.0414, Y 22.4326, Z -6.3333, A 0.000, B 0.000, C 0.000 }
gfCNCPoint4[21588] = {X 326.3723, Y 21.6635, Z -6.3333, A 0.000, B 0.000, C 0.000 }
gfCNCPoint4[21589] = {X 325.7878, Y 20.8284, Z -6.3333, A 0.000, B 0.000, C 0.000 }
gfCNCPoint4[21590] = {X 325.2944, Y 19.9364, Z -6.3333, A 0.000, B 0.000, C 0.000 }
gfCNCPoint4[21591] = {X 321.7736, Y 12.6936, Z -6.3333, A 0.000, B 0.000, C 0.000 }
gfCNCPoint4[21592] = {X 321.6322, Y 12.3894, Z -6.3333, A 0.000, B 0.000, C 0.000 }
gfCNCPoint4[21593] = {X 321.5015, Y 12.0806, Z -6.3333, A 0.000, B 0.000, C 0.000 }
gfCNCPoint4[21594] = {X 321.1058, Y 10.8773, Z -6.3333, A 0.000, B 0.000, C 0.000 }
gfCNCPoint4[21595] = {X 320.8706, Y 9.6327, Z -6.3333, A 0.000, B 0.000, C 0.000 }
gfCNCPoint4[21596] = {X 320.7999, Y 8.3680, Z -6.3333, A 0.000, B 0.000, C 0.000 }
gfCNCPoint4[21597] = {X 320.8950, Y 7.1049, Z -6.3333, A 0.000, B 0.000, C 0.000 }
gfCNCPoint4[21598] = {X 298.7843, Y 7.1049, Z -6.3333, A 0.000, B 0.000, C 0.000 }
gfCNCPoint4[21599] = {X 298.7843, Y 9.5049, Z -6.3333, A 0.000, B 0.000, C 0.000 }
gfCNCPoint4[21600] = {X 297.8291, Y 9.5049, Z -6.3333, A 0.000, B 0.000, C 0.000 }
gfCNCPoint4[21601] = {X 298.1371, Y 10.4755, Z -6.3333, A 0.000, B 0.000, C 0.000 }
gfCNCPoint4[21602] = {X 298.3067, Y 11.4795, Z -6.3333, A 0.000, B 0.000, C 0.000 }
gfCNCPoint4[21603] = {X 298.4763, Y 10.4755, Z -6.3333, A 0.000, B 0.000, C 0.000 }
gfCNCPoint4[21604] = {X 298.7843, Y 9.5049, Z -6.3333, A 0.000, B 0.000, C 0.000 }
gfCNCPoint4[21605] = {X 298.7843, Y 7.1049, Z -6.3333, A 0.000, B 0.000, C 0.000 }
gfCNCPoint4[21606] = {X 233.3038, Y 7.1049, Z -6.3333, A 0.000, B 0.000, C 0.000 }
gfCNCPoint4[21607] = {X 233.3038, Y 11.9049, Z -6.3333, A 0.000, B 0.000, C 0.000 }
gfCNCPoint4[21608] = {X 233.1564, Y 11.9049, Z -6.3333, A 0.000, B 0.000, C 0.000 }
gfCNCPoint4[21609] = {X 233.1594, Y 12.0442, Z -6.3333, A 0.000, B 0.000, C 0.000 }
gfCNCPoint4[21610] = {X 233.1605, Y 12.1835, Z -6.3333, A 0.000, B 0.000, C 0.000 }
gfCNCPoint4[21611] = {X 233.2315, Y 12.0439, Z -6.3333, A 0.000, B 0.000, C 0.000 }
gfCNCPoint4[21612] = {X 233.3038, Y 11.9049, Z -6.3333, A 0.000, B 0.000, C 0.000 }
